LIN {X -0.131,Y -388.858,Z 1048.466,A 0.000,B 0.000,C 90.000,E1 83.856} C_DIS
LIN {X -0.049,Y -379.523,Z 1048.456,A 0.000,B 0.000,C 90.000,E1 82.129} C_DIS
LIN {X -0.037,Y -369.873,Z 1048.447,A 0.000,B 0.000,C 90.000,E1 80.387} C_DIS
LIN {X -0.127,Y -359.894,Z 1048.437,A 0.000,B 0.000,C 90.000,E1 78.634} C_DIS
LIN {X -0.097,Y -346.570,Z 1048.423,A 0.000,B 0.000,C 90.000,E1 76.228} C_DIS
LIN {X 0.098,Y -333.515,Z 1048.410,A 0.000,B 0.000,C 90.000,E1 73.740} C_DIS
LIN {X -0.157,Y -321.006,Z 1048.396,A 0.000,B 0.000,C 90.000,E1 71.275} C_DIS
LIN {X 0.091,Y -308.881,Z 1048.382,A 0.000,B 0.000,C 90.000,E1 68.666} C_DIS
LIN {X 0.079,Y -297.203,Z 1048.367,A 0.000,B 0.000,C 90.000,E1 66.049} C_DIS
LIN {X 0.032,Y -285.773,Z 1048.352,A 0.000,B 0.000,C 90.000,E1 63.384} C_DIS
LIN {X 0.014,Y -275.986,Z 1048.339,A 0.000,B 0.000,C 90.000,E1 61.001} C_DIS
LIN {X 0.100,Y -265.051,Z 1048.323,A 0.000,B 0.000,C 90.000,E1 58.201} C_DIS
LIN {X -0.025,Y -254.368,Z 1048.308,A 0.000,B 0.000,C 90.000,E1 55.388} C_DIS
LIN {X 0.027,Y -242.843,Z 1048.290,A 0.000,B 0.000,C 90.000,E1 52.110} C_DIS
LIN {X 0.019,Y -231.988,Z 1048.271,A 0.000,B 0.000,C 90.000,E1 48.771} C_DIS
LIN {X 0.057,Y -223.046,Z 1048.254,A 0.000,B 0.000,C 90.000,E1 45.729} C_DIS
LIN {X -0.100,Y -214.640,Z 1048.237,A 0.000,B 0.000,C 90.000,E1 42.690} C_DIS
LIN {X 0.029,Y -206.684,Z 1048.220,A 0.000,B 0.000,C 90.000,E1 39.519} C_DIS
LIN {X -0.019,Y -199.257,Z 1048.202,A 0.000,B 0.000,C 90.000,E1 36.343} C_DIS
LIN {X 0.034,Y -192.371,Z 1048.184,A 0.000,B 0.000,C 90.000,E1 33.086} C_DIS
LIN {X 0.034,Y -186.264,Z 1048.166,A 0.000,B 0.000,C 90.000,E1 29.795} C_DIS
LIN {X -0.060,Y -180.873,Z 1048.147,A 0.000,B 0.000,C 90.000,E1 26.488} C_DIS
LIN {X 0.044,Y -176.216,Z 1048.128,A 0.000,B 0.000,C 90.000,E1 23.078} C_DIS
LIN {X -0.014,Y -172.265,Z 1048.109,A 0.000,B 0.000,C 90.000,E1 19.685} C_DIS
LIN {X 0.002,Y -168.389,Z 1048.085,A 0.000,B 0.000,C 90.000,E1 15.371} C_DIS
LIN {X 0.054,Y -165.557,Z 1048.061,A 0.000,B 0.000,C 90.000,E1 11.007} C_DIS
LIN {X 0.024,Y -163.209,Z 1048.022,A 0.000,B 0.000,C 90.000,E1 4.012} C_DIS
LIN {X -0.037,Y -164.388,Z 1047.963,A 0.000,B 0.000,C 90.000,E1 353.394} C_DIS
LIN {X 0.040,Y -167.026,Z 1047.934,A 0.000,B 0.000,C 90.000,E1 348.117} C_DIS
LIN {X -0.032,Y -170.462,Z 1047.910,A 0.000,B 0.000,C 90.000,E1 343.795} C_DIS
LIN {X 0.052,Y -173.950,Z 1047.891,A 0.000,B 0.000,C 90.000,E1 340.315} C_DIS
LIN {X -0.037,Y -178.137,Z 1047.872,A 0.000,B 0.000,C 90.000,E1 336.922} C_DIS
LIN {X 0.030,Y -183.098,Z 1047.853,A 0.000,B 0.000,C 90.000,E1 333.512} C_DIS
LIN {X -0.111,Y -188.880,Z 1047.834,A 0.000,B 0.000,C 90.000,E1 330.205} C_DIS
LIN {X 0.110,Y -195.450,Z 1047.816,A 0.000,B 0.000,C 90.000,E1 326.834} C_DIS
LIN {X -0.044,Y -202.808,Z 1047.798,A 0.000,B 0.000,C 90.000,E1 323.623} C_DIS
LIN {X -0.102,Y -210.701,Z 1047.780,A 0.000,B 0.000,C 90.000,E1 320.436} C_DIS
LIN {X 0.062,Y -220.389,Z 1047.760,A 0.000,B 0.000,C 90.000,E1 316.863} C_DIS
LIN {X 0.075,Y -229.831,Z 1047.743,A 0.000,B 0.000,C 90.000,E1 313.785} C_DIS
LIN {X 0.089,Y -237.669,Z 1047.731,A 0.000,B 0.000,C 90.000,E1 311.515} C_DIS
LIN {X 0.122,Y -246.397,Z 1047.718,A 0.000,B 0.000,C 90.000,E1 309.277} C_DIS
LIN {X 0.137,Y -252.982,Z 1047.710,A 0.000,B 0.000,C 90.000,E1 307.810} C_DIS
LIN {X -0.043,Y -267.797,Z 1047.694,A 0.000,B 0.000,C 90.000,E1 304.978} C_DIS
LIN {X 0.188,Y -286.229,Z 1047.677,A 0.000,B 0.000,C 90.000,E1 301.799} C_DIS
LIN {X -0.040,Y -305.957,Z 1047.660,A 0.000,B 0.000,C 90.000,E1 298.821} C_DIS
LIN {X -0.024,Y -322.578,Z 1047.647,A 0.000,B 0.000,C 90.000,E1 296.539} C_DIS
LIN {X -0.116,Y -332.909,Z 1047.640,A 0.000,B 0.000,C 90.000,E1 295.283} C_DIS
LIN {X -0.126,Y -346.134,Z 1047.632,A 0.000,B 0.000,C 90.000,E1 293.823} C_DIS
LIN {X -0.132,Y -370.998,Z 1047.619,A 0.000,B 0.000,C 90.000,E1 291.408} C_DIS
LIN {X -0.018,Y -390.288,Z 1047.609,A 0.000,B 0.000,C 90.000,E1 289.685} C_DIS
LIN {X 0.047,Y -403.946,Z 1047.603,A 0.000,B 0.000,C 90.000,E1 288.489} C_DIS
LIN {X 0.095,Y -414.628,Z 1047.597,A 0.000,B 0.000,C 90.000,E1 287.528} C_DIS
LIN {X 0.179,Y -422.149,Z 1047.594,A 0.000,B 0.000,C 90.000,E1 286.804} C_DIS
LIN {X -0.051,Y -429.627,Z 1047.589,A 0.000,B 0.000,C 90.000,E1 286.079} C_DIS
LIN {X -0.120,Y -436.988,Z 1047.585,A 0.000,B 0.000,C 90.000,E1 285.300} C_DIS
LIN {X 0.068,Y -444.139,Z 1047.580,A 0.000,B 0.000,C 90.000,E1 284.481} C_DIS
LIN {X -0.013,Y -450.801,Z 1047.576,A 0.000,B 0.000,C 90.000,E1 283.703} C_DIS
LIN {X -0.156,Y -456.953,Z 1047.572,A 0.000,B 0.000,C 90.000,E1 282.939} C_DIS
LIN {X 0.213,Y -462.516,Z 1047.568,A 0.000,B 0.000,C 90.000,E1 282.119} C_DIS
LIN {X 0.084,Y -467.494,Z 1047.563,A 0.000,B 0.000,C 90.000,E1 281.366} C_DIS
LIN {X 0.095,Y -471.818,Z 1047.559,A 0.000,B 0.000,C 90.000,E1 280.602} C_DIS
LIN {X 0.053,Y -475.532,Z 1047.555,A 0.000,B 0.000,C 90.000,E1 279.849} C_DIS
LIN {X 0.255,Y -477.654,Z 1047.552,A 0.000,B 0.000,C 90.000,E1 279.321} C_DIS
LIN {X -0.079,Y -479.547,Z 1047.549,A 0.000,B 0.000,C 90.000,E1 278.859} C_DIS
LIN {X -0.183,Y -482.701,Z 1047.544,A 0.000,B 0.000,C 90.000,E1 277.871} C_DIS
LIN {X -0.016,Y -484.005,Z 1047.541,A 0.000,B 0.000,C 90.000,E1 277.352} C_DIS
LIN {X 0.164,Y -485.073,Z 1047.538,A 0.000,B 0.000,C 90.000,E1 276.834} C_DIS
LIN {X -0.132,Y -485.850,Z 1047.535,A 0.000,B 0.000,C 90.000,E1 276.372} C_DIS
LIN {X 0.060,Y -486.341,Z 1047.533,A 0.000,B 0.000,C 90.000,E1 275.853} C_DIS
LIN {X 0.257,Y -486.480,Z 1047.530,A 0.000,B 0.000,C 90.000,E1 275.334} C_DIS
LIN {X -0.071,Y -486.178,Z 1047.527,A 0.000,B 0.000,C 90.000,E1 274.878} C_DIS
LIN {X 0.129,Y -485.411,Z 1047.524,A 0.000,B 0.000,C 90.000,E1 274.359} C_DIS
LIN {X -0.159,Y -484.101,Z 1047.522,A 0.000,B 0.000,C 90.000,E1 273.898} C_DIS
LIN {X 0.001,Y -482.154,Z 1047.519,A 0.000,B 0.000,C 90.000,E1 273.383} C_DIS
LIN {X 0.179,Y -479.498,Z 1047.516,A 0.000,B 0.000,C 90.000,E1 272.865} C_DIS
LIN {X -0.163,Y -476.100,Z 1047.513,A 0.000,B 0.000,C 90.000,E1 272.407} C_DIS
LIN {X -0.041,Y -471.794,Z 1047.510,A 0.000,B 0.000,C 90.000,E1 271.892} C_DIS
LIN {X 0.070,Y -466.518,Z 1047.508,A 0.000,B 0.000,C 90.000,E1 271.375} C_DIS
LIN {X -0.007,Y -460.835,Z 1047.505,A 0.000,B 0.000,C 90.000,E1 270.917} C_DIS
LIN {X 0.220,Y -454.718,Z 1047.503,A 0.000,B 0.000,C 90.000,E1 270.458} C_DIS
LIN {X -0.065,Y -448.087,Z 1047.501,A 0.000,B 0.000,C 90.000,E1 270.115} C_DIS
LIN {X 0.112,Y -440.719,Z 1047.499,A 0.000,B 0.000,C 90.000,E1 269.771} C_DIS
LIN {X -0.035,Y -432.780,Z 1047.497,A 0.000,B 0.000,C 90.000,E1 269.542} C_DIS
LIN {X -0.102,Y -424.050,Z 1047.496,A 0.000,B 0.000,C 90.000,E1 269.370} C_DIS
LIN {X -0.035,Y -411.377,Z 1047.495,A 0.000,B 0.000,C 90.000,E1 269.198} C_DIS
LIN {X -0.063,Y -401.436,Z 1047.495,A 0.000,B 0.000,C 90.000,E1 269.141} C_DIS
LIN {X 0.162,Y -392.391,Z 1047.495,A 0.000,B 0.000,C 90.000,E1 269.083} C_DIS
LIN {X 0.049,Y -181.341,Z 1047.495,A 0.000,B 0.000,C 90.000,E1 269.083} C_DIS
LIN {X 0.081,Y -180.907,Z 1047.474,A 0.000,B 0.000,C 90.000,E1 265.355} C_DIS
LIN {X -0.026,Y -180.694,Z 1047.470,A 0.000,B 0.000,C 90.000,E1 264.546} C_DIS
LIN {X 0.052,Y -178.779,Z 1047.442,A 0.000,B 0.000,C 90.000,E1 259.454} C_DIS
LIN {X -0.045,Y -175.825,Z 1047.413,A 0.000,B 0.000,C 90.000,E1 254.393} C_DIS
LIN {X -0.044,Y -172.014,Z 1047.385,A 0.000,B 0.000,C 90.000,E1 249.263} C_DIS
LIN {X -0.068,Y -171.434,Z 1047.380,A 0.000,B 0.000,C 90.000,E1 248.411} C_DIS
LIN {X -0.013,Y -167.670,Z 1047.356,A 0.000,B 0.000,C 90.000,E1 244.076} C_DIS
LIN {X -0.073,Y -166.344,Z 1047.346,A 0.000,B 0.000,C 90.000,E1 242.359} C_DIS
LIN {X -0.080,Y -163.079,Z 1047.327,A 0.000,B 0.000,C 90.000,E1 238.869} C_DIS
LIN {X -0.029,Y -161.020,Z 1047.312,A 0.000,B 0.000,C 90.000,E1 236.215} C_DIS
LIN {X -0.045,Y -157.762,Z 1047.293,A 0.000,B 0.000,C 90.000,E1 232.683} C_DIS
LIN {X 0.019,Y -155.800,Z 1047.278,A 0.000,B 0.000,C 90.000,E1 229.989} C_DIS
LIN {X 0.073,Y -152.052,Z 1047.253,A 0.000,B 0.000,C 90.000,E1 225.486} C_DIS
LIN {X -0.020,Y -150.303,Z 1047.238,A 0.000,B 0.000,C 90.000,E1 222.813} C_DIS
LIN {X 0.016,Y -147.048,Z 1047.213,A 0.000,B 0.000,C 90.000,E1 218.257} C_DIS
LIN {X 0.008,Y -145.627,Z 1047.197,A 0.000,B 0.000,C 90.000,E1 215.518} C_DIS
LIN {X 0.007,Y -143.010,Z 1047.172,A 0.000,B 0.000,C 90.000,E1 210.924} C_DIS
LIN {X -0.062,Y -141.637,Z 1047.151,A 0.000,B 0.000,C 90.000,E1 207.257} C_DIS
LIN {X -0.011,Y -139.438,Z 1047.115,A 0.000,B 0.000,C 90.000,E1 200.737} C_DIS
LIN {X 0.042,Y -139.170,Z 1047.105,A 0.000,B 0.000,C 90.000,E1 198.852} C_DIS
LIN {X -0.060,Y -138.318,Z 1047.053,A 0.000,B 0.000,C 90.000,E1 189.557} C_DIS
LIN {X -0.052,Y -139.474,Z 1047.006,A 0.000,B 0.000,C 90.000,E1 181.146} C_DIS
LIN {X 0.029,Y -141.050,Z 1046.975,A 0.000,B 0.000,C 90.000,E1 175.527} C_DIS
LIN {X -0.018,Y -142.421,Z 1046.960,A 0.000,B 0.000,C 90.000,E1 172.761} C_DIS
LIN {X 0.044,Y -144.657,Z 1046.934,A 0.000,B 0.000,C 90.000,E1 168.117} C_DIS
LIN {X -0.038,Y -147.853,Z 1046.909,A 0.000,B 0.000,C 90.000,E1 163.559} C_DIS
LIN {X 0.046,Y -150.555,Z 1046.888,A 0.000,B 0.000,C 90.000,E1 159.880} C_DIS
LIN {X -0.015,Y -154.022,Z 1046.868,A 0.000,B 0.000,C 90.000,E1 156.282} C_DIS
LIN {X -0.017,Y -157.438,Z 1046.848,A 0.000,B 0.000,C 90.000,E1 152.692} C_DIS
LIN {X 0.004,Y -161.652,Z 1046.828,A 0.000,B 0.000,C 90.000,E1 149.125} C_DIS
LIN {X 0.021,Y -165.848,Z 1046.809,A 0.000,B 0.000,C 90.000,E1 145.595} C_DIS
LIN {X 0.013,Y -170.823,Z 1046.790,A 0.000,B 0.000,C 90.000,E1 142.110} C_DIS
LIN {X -0.071,Y -175.692,Z 1046.770,A 0.000,B 0.000,C 90.000,E1 138.690} C_DIS
LIN {X 0.053,Y -181.305,Z 1046.751,A 0.000,B 0.000,C 90.000,E1 135.243} C_DIS
LIN {X -0.075,Y -186.786,Z 1046.733,A 0.000,B 0.000,C 90.000,E1 131.919} C_DIS
LIN {X -0.005,Y -191.379,Z 1046.719,A 0.000,B 0.000,C 90.000,E1 129.402} C_DIS
LIN {X -0.055,Y -197.607,Z 1046.700,A 0.000,B 0.000,C 90.000,E1 125.931} C_DIS
LIN {X 0.103,Y -197.923,Z 1046.699,A 0.000,B 0.000,C 90.000,E1 125.724} C_DIS
LIN {X 0.116,Y -304.006,Z 1046.699,A 0.000,B 0.000,C 90.000,E1 125.724} C_DIS
LIN {X 0.033,Y -305.067,Z 1046.698,A 0.000,B 0.000,C 90.000,E1 125.724} C_DIS
LIN {X -0.019,Y -310.030,Z 1046.697,A 0.000,B 0.000,C 90.000,E1 125.518} C_DIS
LIN {X -0.072,Y -312.622,Z 1046.696,A 0.000,B 0.000,C 90.000,E1 125.311} C_DIS
LIN {X -0.036,Y -316.422,Z 1046.693,A 0.000,B 0.000,C 90.000,E1 124.818} C_DIS
LIN {X 0.019,Y -318.184,Z 1046.692,A 0.000,B 0.000,C 90.000,E1 124.485} C_DIS
LIN {X -0.188,Y -319.561,Z 1046.690,A 0.000,B 0.000,C 90.000,E1 124.199} C_DIS
LIN {X 0.022,Y -332.011,Z 1046.670,A 0.000,B 0.000,C 90.000,E1 120.669} C_DIS
LIN {X -0.149,Y -343.638,Z 1046.655,A 0.000,B 0.000,C 90.000,E1 117.897} C_DIS
LIN {X -0.168,Y -356.702,Z 1046.640,A 0.000,B 0.000,C 90.000,E1 115.155} C_DIS
LIN {X -0.193,Y -369.617,Z 1046.626,A 0.000,B 0.000,C 90.000,E1 112.770} C_DIS
LIN {X -0.183,Y -383.852,Z 1046.613,A 0.000,B 0.000,C 90.000,E1 110.429} C_DIS
LIN {X -0.076,Y -399.507,Z 1046.601,A 0.000,B 0.000,C 90.000,E1 108.127} C_DIS
LIN {X -0.086,Y -416.693,Z 1046.588,A 0.000,B 0.000,C 90.000,E1 105.898} C_DIS
LIN {X -0.011,Y -435.533,Z 1046.576,A 0.000,B 0.000,C 90.000,E1 103.716} C_DIS
LIN {X 0.048,Y -455.539,Z 1046.565,A 0.000,B 0.000,C 90.000,E1 101.658} C_DIS
LIN {X -0.173,Y -468.201,Z 1046.558,A 0.000,B 0.000,C 90.000,E1 100.489} C_DIS
LIN {X -0.225,Y -470.121,Z 1046.557,A 0.000,B 0.000,C 90.000,E1 100.254} C_DIS
LIN {X 0.188,Y -471.578,Z 1046.555,A 0.000,B 0.000,C 90.000,E1 99.962} C_DIS
LIN {X -0.181,Y -473.559,Z 1046.553,A 0.000,B 0.000,C 90.000,E1 99.500} C_DIS
LIN {X 0.002,Y -474.416,Z 1046.550,A 0.000,B 0.000,C 90.000,E1 98.973} C_DIS
LIN {X 0.121,Y -474.297,Z 1046.547,A 0.000,B 0.000,C 90.000,E1 98.454} C_DIS
LIN {X -0.220,Y -473.191,Z 1046.544,A 0.000,B 0.000,C 90.000,E1 97.992} C_DIS
LIN {X 0.110,Y -472.216,Z 1046.543,A 0.000,B 0.000,C 90.000,E1 97.701} C_DIS
LIN {X -0.030,Y -470.902,Z 1046.542,A 0.000,B 0.000,C 90.000,E1 97.466} C_DIS
LIN {X 0.025,Y -458.510,Z 1046.532,A 0.000,B 0.000,C 90.000,E1 95.682} C_DIS
LIN {X 0.035,Y -444.230,Z 1046.520,A 0.000,B 0.000,C 90.000,E1 93.612} C_DIS
LIN {X 0.127,Y -430.922,Z 1046.508,A 0.000,B 0.000,C 90.000,E1 91.489} C_DIS
LIN {X 0.104,Y -415.490,Z 1046.493,A 0.000,B 0.000,C 90.000,E1 88.797} C_DIS
LIN {X -0.121,Y -405.344,Z 1046.483,A 0.000,B 0.000,C 90.000,E1 86.906} C_DIS
LIN {X -0.103,Y -394.835,Z 1046.472,A 0.000,B 0.000,C 90.000,E1 84.951} C_DIS
LIN {X 0.092,Y -385.623,Z 1046.462,A 0.000,B 0.000,C 90.000,E1 83.223} C_DIS
LIN {X 0.158,Y -376.191,Z 1046.453,A 0.000,B 0.000,C 90.000,E1 81.489} C_DIS
LIN {X 0.109,Y -366.399,Z 1046.443,A 0.000,B 0.000,C 90.000,E1 79.746} C_DIS
LIN {X -0.046,Y -356.389,Z 1046.433,A 0.000,B 0.000,C 90.000,E1 77.993} C_DIS
LIN {X -0.025,Y -343.128,Z 1046.420,A 0.000,B 0.000,C 90.000,E1 75.574} C_DIS
LIN {X -0.077,Y -327.078,Z 1046.403,A 0.000,B 0.000,C 90.000,E1 72.489} C_DIS
LIN {X 0.024,Y -314.747,Z 1046.389,A 0.000,B 0.000,C 90.000,E1 69.934} C_DIS
LIN {X -0.164,Y -301.401,Z 1046.372,A 0.000,B 0.000,C 90.000,E1 67.050} C_DIS
LIN {X 0.037,Y -289.864,Z 1046.358,A 0.000,B 0.000,C 90.000,E1 64.357} C_DIS
LIN {X 0.101,Y -280.007,Z 1046.344,A 0.000,B 0.000,C 90.000,E1 61.975} C_DIS
LIN {X 0.148,Y -268.942,Z 1046.329,A 0.000,B 0.000,C 90.000,E1 59.203} C_DIS
LIN {X 0.078,Y -259.487,Z 1046.315,A 0.000,B 0.000,C 90.000,E1 56.755} C_DIS
LIN {X -0.034,Y -248.987,Z 1046.299,A 0.000,B 0.000,C 90.000,E1 53.909} C_DIS
LIN {X 0.011,Y -237.704,Z 1046.281,A 0.000,B 0.000,C 90.000,E1 50.598} C_DIS
LIN {X -0.015,Y -227.230,Z 1046.262,A 0.000,B 0.000,C 90.000,E1 47.229} C_DIS
LIN {X -0.083,Y -218.586,Z 1046.245,A 0.000,B 0.000,C 90.000,E1 44.190} C_DIS
LIN {X -0.035,Y -210.398,Z 1046.228,A 0.000,B 0.000,C 90.000,E1 41.067} C_DIS
LIN {X 0.013,Y -202.682,Z 1046.211,A 0.000,B 0.000,C 90.000,E1 37.890} C_DIS
LIN {X -0.053,Y -195.526,Z 1046.193,A 0.000,B 0.000,C 90.000,E1 34.692} C_DIS
LIN {X 0.059,Y -190.552,Z 1046.179,A 0.000,B 0.000,C 90.000,E1 32.212} C_DIS
LIN {X -0.076,Y -184.618,Z 1046.161,A 0.000,B 0.000,C 90.000,E1 28.949} C_DIS
LIN {X -0.045,Y -179.416,Z 1046.142,A 0.000,B 0.000,C 90.000,E1 25.591} C_DIS
LIN {X -0.051,Y -174.963,Z 1046.123,A 0.000,B 0.000,C 90.000,E1 22.206} C_DIS
LIN {X -0.037,Y -171.220,Z 1046.104,A 0.000,B 0.000,C 90.000,E1 18.779} C_DIS
LIN {X -0.097,Y -167.530,Z 1046.080,A 0.000,B 0.000,C 90.000,E1 14.481} C_DIS
LIN {X 0.055,Y -165.004,Z 1046.056,A 0.000,B 0.000,C 90.000,E1 10.074} C_DIS
LIN {X -0.038,Y -162.952,Z 1046.017,A 0.000,B 0.000,C 90.000,E1 3.094} C_DIS
LIN {X -0.042,Y -164.283,Z 1045.963,A 0.000,B 0.000,C 90.000,E1 353.394} C_DIS
LIN {X 0.031,Y -166.926,Z 1045.934,A 0.000,B 0.000,C 90.000,E1 348.117} C_DIS
LIN {X -0.044,Y -170.370,Z 1045.910,A 0.000,B 0.000,C 90.000,E1 343.795} C_DIS
LIN {X 0.037,Y -173.856,Z 1045.891,A 0.000,B 0.000,C 90.000,E1 340.315} C_DIS
LIN {X -0.054,Y -178.038,Z 1045.872,A 0.000,B 0.000,C 90.000,E1 336.922} C_DIS
LIN {X 0.010,Y -183.000,Z 1045.853,A 0.000,B 0.000,C 90.000,E1 333.512} C_DIS
LIN {X 0.125,Y -188.808,Z 1045.834,A 0.000,B 0.000,C 90.000,E1 330.127} C_DIS
LIN {X 0.084,Y -195.389,Z 1045.816,A 0.000,B 0.000,C 90.000,E1 326.834} C_DIS
LIN {X -0.072,Y -202.763,Z 1045.798,A 0.000,B 0.000,C 90.000,E1 323.623} C_DIS
LIN {X -0.132,Y -210.641,Z 1045.780,A 0.000,B 0.000,C 90.000,E1 320.436} C_DIS
LIN {X 0.028,Y -220.328,Z 1045.760,A 0.000,B 0.000,C 90.000,E1 316.863} C_DIS
LIN {X 0.038,Y -229.752,Z 1045.743,A 0.000,B 0.000,C 90.000,E1 313.785} C_DIS
LIN {X 0.049,Y -237.577,Z 1045.731,A 0.000,B 0.000,C 90.000,E1 311.515} C_DIS
LIN {X 0.080,Y -246.318,Z 1045.718,A 0.000,B 0.000,C 90.000,E1 309.277} C_DIS
LIN {X 0.092,Y -252.891,Z 1045.710,A 0.000,B 0.000,C 90.000,E1 307.810} C_DIS
LIN {X 0.061,Y -267.723,Z 1045.694,A 0.000,B 0.000,C 90.000,E1 304.945} C_DIS
LIN {X 0.132,Y -286.216,Z 1045.677,A 0.000,B 0.000,C 90.000,E1 301.799} C_DIS
LIN {X -0.099,Y -305.987,Z 1045.660,A 0.000,B 0.000,C 90.000,E1 298.821} C_DIS
LIN {X -0.085,Y -322.667,Z 1045.647,A 0.000,B 0.000,C 90.000,E1 296.539} C_DIS
LIN {X 0.073,Y -335.551,Z 1045.639,A 0.000,B 0.000,C 90.000,E1 294.951} C_DIS
LIN {X -0.083,Y -349.150,Z 1045.631,A 0.000,B 0.000,C 90.000,E1 293.515} C_DIS
LIN {X 0.198,Y -379.470,Z 1045.615,A 0.000,B 0.000,C 90.000,E1 290.610} C_DIS
LIN {X -0.047,Y -395.869,Z 1045.607,A 0.000,B 0.000,C 90.000,E1 289.214} C_DIS
LIN {X 0.126,Y -406.758,Z 1045.601,A 0.000,B 0.000,C 90.000,E1 288.236} C_DIS
LIN {X 0.173,Y -414.756,Z 1045.597,A 0.000,B 0.000,C 90.000,E1 287.511} C_DIS
LIN {X -0.038,Y -422.492,Z 1045.593,A 0.000,B 0.000,C 90.000,E1 286.804} C_DIS
LIN {X 0.076,Y -429.992,Z 1045.589,A 0.000,B 0.000,C 90.000,E1 286.024} C_DIS
LIN {X 0.172,Y -439.780,Z 1045.583,A 0.000,B 0.000,C 90.000,E1 284.954} C_DIS
LIN {X 0.056,Y -446.756,Z 1045.579,A 0.000,B 0.000,C 90.000,E1 284.175} C_DIS
LIN {X -0.120,Y -453.230,Z 1045.574,A 0.000,B 0.000,C 90.000,E1 283.411} C_DIS
LIN {X 0.213,Y -459.118,Z 1045.570,A 0.000,B 0.000,C 90.000,E1 282.591} C_DIS
LIN {X 0.149,Y -464.473,Z 1045.566,A 0.000,B 0.000,C 90.000,E1 281.827} C_DIS
LIN {X 0.042,Y -469.238,Z 1045.562,A 0.000,B 0.000,C 90.000,E1 281.074} C_DIS
LIN {X 0.064,Y -473.345,Z 1045.557,A 0.000,B 0.000,C 90.000,E1 280.310} C_DIS
LIN {X 0.039,Y -476.856,Z 1045.553,A 0.000,B 0.000,C 90.000,E1 279.557} C_DIS
LIN {X 0.043,Y -479.763,Z 1045.549,A 0.000,B 0.000,C 90.000,E1 278.803} C_DIS
LIN {X -0.056,Y -482.894,Z 1045.543,A 0.000,B 0.000,C 90.000,E1 277.814} C_DIS
LIN {X 0.113,Y -484.162,Z 1045.541,A 0.000,B 0.000,C 90.000,E1 277.296} C_DIS
LIN {X -0.187,Y -485.227,Z 1045.538,A 0.000,B 0.000,C 90.000,E1 276.834} C_DIS
LIN {X 0.001,Y -486.001,Z 1045.535,A 0.000,B 0.000,C 90.000,E1 276.315} C_DIS
LIN {X 0.194,Y -486.460,Z 1045.532,A 0.000,B 0.000,C 90.000,E1 275.796} C_DIS
LIN {X -0.092,Y -486.565,Z 1045.530,A 0.000,B 0.000,C 90.000,E1 275.334} C_DIS
LIN {X 0.065,Y -486.236,Z 1045.527,A 0.000,B 0.000,C 90.000,E1 274.821} C_DIS
LIN {X -0.217,Y -485.456,Z 1045.524,A 0.000,B 0.000,C 90.000,E1 274.359} C_DIS
LIN {X -0.022,Y -484.097,Z 1045.521,A 0.000,B 0.000,C 90.000,E1 273.841} C_DIS
LIN {X 0.138,Y -482.101,Z 1045.519,A 0.000,B 0.000,C 90.000,E1 273.326} C_DIS
LIN {X -0.163,Y -479.410,Z 1045.516,A 0.000,B 0.000,C 90.000,E1 272.865} C_DIS
LIN {X 0.143,Y -477.802,Z 1045.514,A 0.000,B 0.000,C 90.000,E1 272.579} C_DIS
LIN {X -0.203,Y -473.886,Z 1045.512,A 0.000,B 0.000,C 90.000,E1 272.121} C_DIS
LIN {X -0.080,Y -469.073,Z 1045.509,A 0.000,B 0.000,C 90.000,E1 271.604} C_DIS
LIN {X 0.187,Y -463.534,Z 1045.506,A 0.000,B 0.000,C 90.000,E1 271.088} C_DIS
LIN {X -0.157,Y -457.703,Z 1045.504,A 0.000,B 0.000,C 90.000,E1 270.688} C_DIS
LIN {X -0.161,Y -451.404,Z 1045.501,A 0.000,B 0.000,C 90.000,E1 270.286} C_DIS
LIN {X 0.157,Y -447.914,Z 1045.500,A 0.000,B 0.000,C 90.000,E1 270.057} C_DIS
LIN {X -0.092,Y -440.528,Z 1045.499,A 0.000,B 0.000,C 90.000,E1 269.771} C_DIS
LIN {X -0.157,Y -436.976,Z 1045.498,A 0.000,B 0.000,C 90.000,E1 269.656} C_DIS
LIN {X -0.006,Y -428.802,Z 1045.497,A 0.000,B 0.000,C 90.000,E1 269.427} C_DIS
LIN {X 0.200,Y -420.015,Z 1045.496,A 0.000,B 0.000,C 90.000,E1 269.255} C_DIS
LIN {X -0.133,Y -411.331,Z 1045.495,A 0.000,B 0.000,C 90.000,E1 269.198} C_DIS
LIN {X -0.158,Y -401.181,Z 1045.495,A 0.000,B 0.000,C 90.000,E1 269.141} C_DIS
LIN {X 0.129,Y -395.536,Z 1045.495,A 0.000,B 0.000,C 90.000,E1 269.083} C_DIS
LIN {X 0.033,Y -181.340,Z 1045.495,A 0.000,B 0.000,C 90.000,E1 269.083} C_DIS
LIN {X 0.040,Y -180.906,Z 1045.474,A 0.000,B 0.000,C 90.000,E1 265.355} C_DIS
LIN {X -0.066,Y -180.688,Z 1045.470,A 0.000,B 0.000,C 90.000,E1 264.546} C_DIS
LIN {X 0.012,Y -178.772,Z 1045.441,A 0.000,B 0.000,C 90.000,E1 259.454} C_DIS
LIN {X 0.084,Y -175.818,Z 1045.413,A 0.000,B 0.000,C 90.000,E1 254.338} C_DIS
LIN {X 0.078,Y -172.006,Z 1045.385,A 0.000,B 0.000,C 90.000,E1 249.209} C_DIS
LIN {X 0.052,Y -171.423,Z 1045.380,A 0.000,B 0.000,C 90.000,E1 248.358} C_DIS
LIN {X -0.052,Y -167.661,Z 1045.356,A 0.000,B 0.000,C 90.000,E1 244.076} C_DIS
LIN {X 0.036,Y -166.330,Z 1045.346,A 0.000,B 0.000,C 90.000,E1 242.308} C_DIS
LIN {X 0.022,Y -163.068,Z 1045.327,A 0.000,B 0.000,C 90.000,E1 238.820} C_DIS
LIN {X -0.067,Y -161.007,Z 1045.312,A 0.000,B 0.000,C 90.000,E1 236.215} C_DIS
LIN {X 0.044,Y -157.751,Z 1045.292,A 0.000,B 0.000,C 90.000,E1 232.637} C_DIS
LIN {X -0.018,Y -155.789,Z 1045.278,A 0.000,B 0.000,C 90.000,E1 229.989} C_DIS
LIN {X 0.037,Y -152.043,Z 1045.253,A 0.000,B 0.000,C 90.000,E1 225.486} C_DIS
LIN {X 0.054,Y -150.292,Z 1045.238,A 0.000,B 0.000,C 90.000,E1 222.771} C_DIS
LIN {X -0.020,Y -147.040,Z 1045.213,A 0.000,B 0.000,C 90.000,E1 218.257} C_DIS
LIN {X -0.027,Y -145.620,Z 1045.197,A 0.000,B 0.000,C 90.000,E1 215.518} C_DIS
LIN {X -0.029,Y -143.004,Z 1045.172,A 0.000,B 0.000,C 90.000,E1 210.924} C_DIS
LIN {X 0.029,Y -141.630,Z 1045.151,A 0.000,B 0.000,C 90.000,E1 207.206} C_DIS
LIN {X -0.045,Y -139.435,Z 1045.115,A 0.000,B 0.000,C 90.000,E1 200.737} C_DIS
LIN {X 0.009,Y -139.167,Z 1045.105,A 0.000,B 0.000,C 90.000,E1 198.852} C_DIS
LIN {X 0.042,Y -138.316,Z 1045.053,A 0.000,B 0.000,C 90.000,E1 189.500} C_DIS
LIN {X 0.053,Y -139.475,Z 1045.006,A 0.000,B 0.000,C 90.000,E1 181.088} C_DIS
LIN {X -0.006,Y -141.056,Z 1044.975,A 0.000,B 0.000,C 90.000,E1 175.527} C_DIS
LIN {X -0.052,Y -142.429,Z 1044.960,A 0.000,B 0.000,C 90.000,E1 172.761} C_DIS
LIN {X 0.009,Y -144.665,Z 1044.934,A 0.000,B 0.000,C 90.000,E1 168.117} C_DIS
LIN {X -0.007,Y -147.250,Z 1044.914,A 0.000,B 0.000,C 90.000,E1 164.448} C_DIS
LIN {X 0.010,Y -150.567,Z 1044.888,A 0.000,B 0.000,C 90.000,E1 159.880} C_DIS
LIN {X 0.090,Y -154.036,Z 1044.868,A 0.000,B 0.000,C 90.000,E1 156.230} C_DIS
LIN {X 0.018,Y -157.452,Z 1044.848,A 0.000,B 0.000,C 90.000,E1 152.666} C_DIS
LIN {X -0.034,Y -161.670,Z 1044.828,A 0.000,B 0.000,C 90.000,E1 149.125} C_DIS
LIN {X -0.017,Y -165.866,Z 1044.809,A 0.000,B 0.000,C 90.000,E1 145.595} C_DIS
LIN {X -0.025,Y -170.843,Z 1044.789,A 0.000,B 0.000,C 90.000,E1 142.110} C_DIS
LIN {X 0.021,Y -175.712,Z 1044.770,A 0.000,B 0.000,C 90.000,E1 138.647} C_DIS
LIN {X 0.013,Y -181.324,Z 1044.751,A 0.000,B 0.000,C 90.000,E1 135.243} C_DIS
LIN {X 0.007,Y -186.809,Z 1044.733,A 0.000,B 0.000,C 90.000,E1 131.881} C_DIS
LIN {X -0.047,Y -191.398,Z 1044.719,A 0.000,B 0.000,C 90.000,E1 129.402} C_DIS
LIN {X 0.063,Y -197.631,Z 1044.699,A 0.000,B 0.000,C 90.000,E1 125.884} C_DIS
LIN {X -0.034,Y -197.843,Z 1044.699,A 0.000,B 0.000,C 90.000,E1 125.804} C_DIS
LIN {X -0.099,Y -304.134,Z 1044.699,A 0.000,B 0.000,C 90.000,E1 125.804} C_DIS
LIN {X 0.073,Y -310.224,Z 1044.697,A 0.000,B 0.000,C 90.000,E1 125.518} C_DIS
LIN {X -0.140,Y -312.986,Z 1044.696,A 0.000,B 0.000,C 90.000,E1 125.311} C_DIS
LIN {X 0.014,Y -316.737,Z 1044.693,A 0.000,B 0.000,C 90.000,E1 124.771} C_DIS
LIN {X -0.011,Y -318.393,Z 1044.691,A 0.000,B 0.000,C 90.000,E1 124.452} C_DIS
LIN {X 0.120,Y -320.761,Z 1044.688,A 0.000,B 0.000,C 90.000,E1 123.785} C_DIS
LIN {X 0.147,Y -330.924,Z 1044.672,A 0.000,B 0.000,C 90.000,E1 120.924} C_DIS
LIN {X -0.051,Y -342.412,Z 1044.656,A 0.000,B 0.000,C 90.000,E1 118.153} C_DIS
LIN {X -0.106,Y -355.333,Z 1044.641,A 0.000,B 0.000,C 90.000,E1 115.412} C_DIS
LIN {X -0.019,Y -368.109,Z 1044.628,A 0.000,B 0.000,C 90.000,E1 113.003} C_DIS
LIN {X -0.049,Y -382.194,Z 1044.615,A 0.000,B 0.000,C 90.000,E1 110.663} C_DIS
LIN {X 0.014,Y -397.688,Z 1044.602,A 0.000,B 0.000,C 90.000,E1 108.362} C_DIS
LIN {X -0.041,Y -414.699,Z 1044.590,A 0.000,B 0.000,C 90.000,E1 106.134} C_DIS
LIN {X 0.087,Y -433.353,Z 1044.578,A 0.000,B 0.000,C 90.000,E1 103.939} C_DIS
LIN {X -0.020,Y -453.293,Z 1044.566,A 0.000,B 0.000,C 90.000,E1 101.883} C_DIS
LIN {X 0.060,Y -468.424,Z 1044.558,A 0.000,B 0.000,C 90.000,E1 100.433} C_DIS
LIN {X -0.017,Y -470.305,Z 1044.557,A 0.000,B 0.000,C 90.000,E1 100.197} C_DIS
LIN {X -0.094,Y -471.729,Z 1044.555,A 0.000,B 0.000,C 90.000,E1 99.962} C_DIS
LIN {X 0.004,Y -473.627,Z 1044.552,A 0.000,B 0.000,C 90.000,E1 99.443} C_DIS
LIN {X 0.188,Y -474.418,Z 1044.550,A 0.000,B 0.000,C 90.000,E1 98.916} C_DIS
LIN {X -0.160,Y -474.236,Z 1044.547,A 0.000,B 0.000,C 90.000,E1 98.454} C_DIS
LIN {X -0.033,Y -473.061,Z 1044.544,A 0.000,B 0.000,C 90.000,E1 97.936} C_DIS
LIN {X -0.170,Y -472.045,Z 1044.543,A 0.000,B 0.000,C 90.000,E1 97.701} C_DIS
LIN {X 0.157,Y -470.681,Z 1044.541,A 0.000,B 0.000,C 90.000,E1 97.409} C_DIS
LIN {X 0.204,Y -458.264,Z 1044.531,A 0.000,B 0.000,C 90.000,E1 95.625} C_DIS
LIN {X 0.015,Y -445.759,Z 1044.521,A 0.000,B 0.000,C 90.000,E1 93.841} C_DIS
LIN {X -0.036,Y -433.918,Z 1044.511,A 0.000,B 0.000,C 90.000,E1 92.007} C_DIS
LIN {X 0.153,Y -416.757,Z 1044.495,A 0.000,B 0.000,C 90.000,E1 89.026} C_DIS
LIN {X -0.050,Y -406.599,Z 1044.484,A 0.000,B 0.000,C 90.000,E1 87.135} C_DIS
LIN {X -0.072,Y -397.653,Z 1044.475,A 0.000,B 0.000,C 90.000,E1 85.469} C_DIS
LIN {X 0.173,Y -388.511,Z 1044.465,A 0.000,B 0.000,C 90.000,E1 83.742} C_DIS
LIN {X -0.085,Y -379.177,Z 1044.456,A 0.000,B 0.000,C 90.000,E1 82.064} C_DIS
LIN {X -0.131,Y -369.477,Z 1044.446,A 0.000,B 0.000,C 90.000,E1 80.330} C_DIS
LIN {X 0.126,Y -359.515,Z 1044.436,A 0.000,B 0.000,C 90.000,E1 78.522} C_DIS
LIN {X -0.134,Y -347.896,Z 1044.425,A 0.000,B 0.000,C 90.000,E1 76.464} C_DIS
LIN {X 0.095,Y -334.795,Z 1044.411,A 0.000,B 0.000,C 90.000,E1 73.976} C_DIS
LIN {X -0.126,Y -322.231,Z 1044.397,A 0.000,B 0.000,C 90.000,E1 71.511} C_DIS
LIN {X 0.072,Y -308.555,Z 1044.381,A 0.000,B 0.000,C 90.000,E1 68.592} C_DIS
LIN {X 0.059,Y -298.314,Z 1044.368,A 0.000,B 0.000,C 90.000,E1 66.305} C_DIS
LIN {X 0.036,Y -286.843,Z 1044.354,A 0.000,B 0.000,C 90.000,E1 63.640} C_DIS
LIN {X 0.039,Y -277.003,Z 1044.340,A 0.000,B 0.000,C 90.000,E1 61.257} C_DIS
LIN {X 0.012,Y -266.020,Z 1044.325,A 0.000,B 0.000,C 90.000,E1 58.486} C_DIS
LIN {X -0.089,Y -255.303,Z 1044.309,A 0.000,B 0.000,C 90.000,E1 55.674} C_DIS
LIN {X -0.008,Y -243.666,Z 1044.291,A 0.000,B 0.000,C 90.000,E1 52.396} C_DIS
LIN {X 0.008,Y -232.742,Z 1044.273,A 0.000,B 0.000,C 90.000,E1 49.057} C_DIS
LIN {X 0.005,Y -222.645,Z 1044.254,A 0.000,B 0.000,C 90.000,E1 45.648} C_DIS
LIN {X -0.002,Y -214.193,Z 1044.236,A 0.000,B 0.000,C 90.000,E1 42.567} C_DIS
LIN {X -0.040,Y -206.257,Z 1044.219,A 0.000,B 0.000,C 90.000,E1 39.439} C_DIS
LIN {X 0.061,Y -198.801,Z 1044.201,A 0.000,B 0.000,C 90.000,E1 36.217} C_DIS
LIN {X 0.104,Y -191.906,Z 1044.183,A 0.000,B 0.000,C 90.000,E1 32.959} C_DIS
LIN {X 0.093,Y -185.801,Z 1044.165,A 0.000,B 0.000,C 90.000,E1 29.667} C_DIS
LIN {X -0.013,Y -180.423,Z 1044.146,A 0.000,B 0.000,C 90.000,E1 26.360} C_DIS
LIN {X 0.077,Y -175.788,Z 1044.128,A 0.000,B 0.000,C 90.000,E1 22.950} C_DIS
LIN {X -0.051,Y -171.878,Z 1044.109,A 0.000,B 0.000,C 90.000,E1 19.577} C_DIS
LIN {X 0.006,Y -168.013,Z 1044.085,A 0.000,B 0.000,C 90.000,E1 15.245} C_DIS
LIN {X 0.009,Y -165.253,Z 1044.061,A 0.000,B 0.000,C 90.000,E1 10.894} C_DIS
LIN {X 0.019,Y -163.106,Z 1044.026,A 0.000,B 0.000,C 90.000,E1 4.759} C_DIS
LIN {X -0.046,Y -164.184,Z 1043.963,A 0.000,B 0.000,C 90.000,E1 353.394} C_DIS
LIN {X 0.023,Y -166.839,Z 1043.934,A 0.000,B 0.000,C 90.000,E1 348.117} C_DIS
LIN {X -0.054,Y -170.285,Z 1043.910,A 0.000,B 0.000,C 90.000,E1 343.795} C_DIS
LIN {X 0.025,Y -173.762,Z 1043.891,A 0.000,B 0.000,C 90.000,E1 340.315} C_DIS
LIN {X -0.069,Y -177.940,Z 1043.872,A 0.000,B 0.000,C 90.000,E1 336.922} C_DIS
LIN {X -0.008,Y -182.902,Z 1043.853,A 0.000,B 0.000,C 90.000,E1 333.512} C_DIS
LIN {X 0.103,Y -188.732,Z 1043.834,A 0.000,B 0.000,C 90.000,E1 330.127} C_DIS
LIN {X 0.060,Y -195.343,Z 1043.816,A 0.000,B 0.000,C 90.000,E1 326.834} C_DIS
LIN {X -0.098,Y -202.715,Z 1043.798,A 0.000,B 0.000,C 90.000,E1 323.623} C_DIS
LIN {X 0.136,Y -210.583,Z 1043.780,A 0.000,B 0.000,C 90.000,E1 320.356} C_DIS
LIN {X -0.004,Y -220.266,Z 1043.760,A 0.000,B 0.000,C 90.000,E1 316.863} C_DIS
LIN {X 0.003,Y -229.681,Z 1043.743,A 0.000,B 0.000,C 90.000,E1 313.785} C_DIS
LIN {X -0.023,Y -238.896,Z 1043.729,A 0.000,B 0.000,C 90.000,E1 311.148} C_DIS
LIN {X 0.039,Y -246.247,Z 1043.718,A 0.000,B 0.000,C 90.000,E1 309.277} C_DIS
LIN {X 0.049,Y -252.798,Z 1043.710,A 0.000,B 0.000,C 90.000,E1 307.810} C_DIS
LIN {X -0.044,Y -265.707,Z 1043.696,A 0.000,B 0.000,C 90.000,E1 305.311} C_DIS
LIN {X 0.126,Y -284.083,Z 1043.679,A 0.000,B 0.000,C 90.000,E1 302.133} C_DIS
LIN {X -0.027,Y -303.749,Z 1043.662,A 0.000,B 0.000,C 90.000,E1 299.127} C_DIS
LIN {X 0.081,Y -320.261,Z 1043.649,A 0.000,B 0.000,C 90.000,E1 296.821} C_DIS
LIN {X -0.111,Y -333.020,Z 1043.640,A 0.000,B 0.000,C 90.000,E1 295.283} C_DIS
LIN {X 0.062,Y -346.539,Z 1043.632,A 0.000,B 0.000,C 90.000,E1 293.770} C_DIS
LIN {X -0.145,Y -371.275,Z 1043.619,A 0.000,B 0.000,C 90.000,E1 291.408} C_DIS
LIN {X 0.217,Y -390.729,Z 1043.609,A 0.000,B 0.000,C 90.000,E1 289.631} C_DIS
LIN {X -0.066,Y -404.295,Z 1043.603,A 0.000,B 0.000,C 90.000,E1 288.489} C_DIS
LIN {X 0.089,Y -414.896,Z 1043.597,A 0.000,B 0.000,C 90.000,E1 287.511} C_DIS
LIN {X -0.193,Y -422.743,Z 1043.593,A 0.000,B 0.000,C 90.000,E1 286.804} C_DIS
LIN {X -0.144,Y -430.260,Z 1043.589,A 0.000,B 0.000,C 90.000,E1 286.024} C_DIS
LIN {X -0.085,Y -440.060,Z 1043.583,A 0.000,B 0.000,C 90.000,E1 284.954} C_DIS
LIN {X 0.231,Y -446.991,Z 1043.579,A 0.000,B 0.000,C 90.000,E1 284.120} C_DIS
LIN {X 0.061,Y -453.423,Z 1043.574,A 0.000,B 0.000,C 90.000,E1 283.355} C_DIS
LIN {X 0.223,Y -461.168,Z 1043.568,A 0.000,B 0.000,C 90.000,E1 282.299} C_DIS
LIN {X 0.182,Y -466.315,Z 1043.564,A 0.000,B 0.000,C 90.000,E1 281.535} C_DIS
LIN {X 0.089,Y -470.853,Z 1043.560,A 0.000,B 0.000,C 90.000,E1 280.782} C_DIS
LIN {X 0.126,Y -474.744,Z 1043.556,A 0.000,B 0.000,C 90.000,E1 280.018} C_DIS
LIN {X 0.110,Y -478.029,Z 1043.552,A 0.000,B 0.000,C 90.000,E1 279.265} C_DIS
LIN {X -0.223,Y -479.926,Z 1043.549,A 0.000,B 0.000,C 90.000,E1 278.803} C_DIS
LIN {X 0.157,Y -483.042,Z 1043.543,A 0.000,B 0.000,C 90.000,E1 277.757} C_DIS
LIN {X -0.152,Y -484.298,Z 1043.540,A 0.000,B 0.000,C 90.000,E1 277.296} C_DIS
LIN {X 0.029,Y -485.352,Z 1043.538,A 0.000,B 0.000,C 90.000,E1 276.777} C_DIS
LIN {X 0.219,Y -486.115,Z 1043.535,A 0.000,B 0.000,C 90.000,E1 276.258} C_DIS
LIN {X -0.071,Y -486.593,Z 1043.532,A 0.000,B 0.000,C 90.000,E1 275.796} C_DIS
LIN {X 0.128,Y -486.665,Z 1043.529,A 0.000,B 0.000,C 90.000,E1 275.277} C_DIS
LIN {X -0.197,Y -486.318,Z 1043.527,A 0.000,B 0.000,C 90.000,E1 274.821} C_DIS
LIN {X 0.005,Y -485.488,Z 1043.524,A 0.000,B 0.000,C 90.000,E1 274.302} C_DIS
LIN {X 0.201,Y -484.116,Z 1043.521,A 0.000,B 0.000,C 90.000,E1 273.784} C_DIS
LIN {X -0.122,Y -482.101,Z 1043.518,A 0.000,B 0.000,C 90.000,E1 273.326} C_DIS
LIN {X 0.222,Y -480.863,Z 1043.517,A 0.000,B 0.000,C 90.000,E1 273.037} C_DIS
LIN {X -0.113,Y -477.766,Z 1043.514,A 0.000,B 0.000,C 90.000,E1 272.579} C_DIS
LIN {X 0.015,Y -473.775,Z 1043.511,A 0.000,B 0.000,C 90.000,E1 272.064} C_DIS
LIN {X 0.136,Y -468.951,Z 1043.509,A 0.000,B 0.000,C 90.000,E1 271.547} C_DIS
LIN {X -0.077,Y -463.433,Z 1043.506,A 0.000,B 0.000,C 90.000,E1 271.088} C_DIS
LIN {X 0.032,Y -457.600,Z 1043.504,A 0.000,B 0.000,C 90.000,E1 270.630} C_DIS
LIN {X 0.053,Y -451.266,Z 1043.501,A 0.000,B 0.000,C 90.000,E1 270.229} C_DIS
LIN {X 0.049,Y -444.376,Z 1043.499,A 0.000,B 0.000,C 90.000,E1 269.885} C_DIS
LIN {X 0.153,Y -440.439,Z 1043.499,A 0.000,B 0.000,C 90.000,E1 269.714} C_DIS
LIN {X 0.026,Y -432.170,Z 1043.497,A 0.000,B 0.000,C 90.000,E1 269.484} C_DIS
LIN {X 0.041,Y -423.424,Z 1043.496,A 0.000,B 0.000,C 90.000,E1 269.312} C_DIS
LIN {X 0.053,Y -415.035,Z 1043.496,A 0.000,B 0.000,C 90.000,E1 269.198} C_DIS
LIN {X -0.017,Y -407.773,Z 1043.495,A 0.000,B 0.000,C 90.000,E1 269.141} C_DIS
LIN {X 0.123,Y -400.048,Z 1043.495,A 0.000,B 0.000,C 90.000,E1 269.083} C_DIS
LIN {X 0.020,Y -393.457,Z 1043.495,A 0.000,B 0.000,C 90.000,E1 269.083} C_DIS
LIN {X -0.014,Y -181.336,Z 1043.495,A 0.000,B 0.000,C 90.000,E1 269.083} C_DIS
LIN {X -0.001,Y -180.906,Z 1043.474,A 0.000,B 0.000,C 90.000,E1 265.355} C_DIS
LIN {X 0.072,Y -180.681,Z 1043.469,A 0.000,B 0.000,C 90.000,E1 264.489} C_DIS
LIN {X -0.029,Y -178.765,Z 1043.441,A 0.000,B 0.000,C 90.000,E1 259.454} C_DIS
LIN {X 0.043,Y -175.811,Z 1043.413,A 0.000,B 0.000,C 90.000,E1 254.338} C_DIS
LIN {X 0.037,Y -171.998,Z 1043.385,A 0.000,B 0.000,C 90.000,E1 249.209} C_DIS
LIN {X 0.012,Y -171.411,Z 1043.380,A 0.000,B 0.000,C 90.000,E1 248.358} C_DIS
LIN {X 0.059,Y -167.650,Z 1043.356,A 0.000,B 0.000,C 90.000,E1 244.024} C_DIS
LIN {X 0.073,Y -166.316,Z 1043.346,A 0.000,B 0.000,C 90.000,E1 242.281} C_DIS
LIN {X 0.067,Y -163.057,Z 1043.327,A 0.000,B 0.000,C 90.000,E1 238.791} C_DIS
LIN {X 0.029,Y -160.993,Z 1043.312,A 0.000,B 0.000,C 90.000,E1 236.167} C_DIS
LIN {X 0.006,Y -157.740,Z 1043.292,A 0.000,B 0.000,C 90.000,E1 232.637} C_DIS
LIN {X -0.056,Y -155.778,Z 1043.278,A 0.000,B 0.000,C 90.000,E1 229.989} C_DIS
LIN {X -0.001,Y -152.033,Z 1043.253,A 0.000,B 0.000,C 90.000,E1 225.486} C_DIS
LIN {X 0.017,Y -150.281,Z 1043.238,A 0.000,B 0.000,C 90.000,E1 222.771} C_DIS
LIN {X -0.056,Y -147.031,Z 1043.212,A 0.000,B 0.000,C 90.000,E1 218.257} C_DIS
LIN {X -0.064,Y -145.612,Z 1043.197,A 0.000,B 0.000,C 90.000,E1 215.518} C_DIS
LIN {X -0.064,Y -142.997,Z 1043.172,A 0.000,B 0.000,C 90.000,E1 210.924} C_DIS
LIN {X -0.007,Y -141.624,Z 1043.151,A 0.000,B 0.000,C 90.000,E1 207.206} C_DIS
LIN {X -0.082,Y -139.432,Z 1043.115,A 0.000,B 0.000,C 90.000,E1 200.737} C_DIS
LIN {X -0.027,Y -139.163,Z 1043.105,A 0.000,B 0.000,C 90.000,E1 198.852} C_DIS
LIN {X 0.010,Y -138.340,Z 1043.058,A 0.000,B 0.000,C 90.000,E1 190.433} C_DIS
LIN {X 0.017,Y -139.477,Z 1043.006,A 0.000,B 0.000,C 90.000,E1 181.088} C_DIS
LIN {X -0.042,Y -141.062,Z 1042.975,A 0.000,B 0.000,C 90.000,E1 175.527} C_DIS
LIN {X 0.053,Y -142.435,Z 1042.960,A 0.000,B 0.000,C 90.000,E1 172.704} C_DIS
LIN {X -0.028,Y -144.674,Z 1042.934,A 0.000,B 0.000,C 90.000,E1 168.117} C_DIS
LIN {X -0.045,Y -147.261,Z 1042.913,A 0.000,B 0.000,C 90.000,E1 164.448} C_DIS
LIN {X -0.027,Y -150.579,Z 1042.888,A 0.000,B 0.000,C 90.000,E1 159.880} C_DIS
LIN {X 0.052,Y -154.050,Z 1042.868,A 0.000,B 0.000,C 90.000,E1 156.230} C_DIS
LIN {X -0.021,Y -157.467,Z 1042.848,A 0.000,B 0.000,C 90.000,E1 152.666} C_DIS
LIN {X 0.066,Y -161.689,Z 1042.828,A 0.000,B 0.000,C 90.000,E1 149.076} C_DIS
LIN {X -0.057,Y -165.883,Z 1042.809,A 0.000,B 0.000,C 90.000,E1 145.595} C_DIS
LIN {X -0.067,Y -170.863,Z 1042.789,A 0.000,B 0.000,C 90.000,E1 142.110} C_DIS
LIN {X -0.020,Y -175.733,Z 1042.770,A 0.000,B 0.000,C 90.000,E1 138.647} C_DIS
LIN {X -0.030,Y -181.343,Z 1042.751,A 0.000,B 0.000,C 90.000,E1 135.243} C_DIS
LIN {X 0.104,Y -186.833,Z 1042.733,A 0.000,B 0.000,C 90.000,E1 131.838} C_DIS
LIN {X 0.058,Y -191.420,Z 1042.719,A 0.000,B 0.000,C 90.000,E1 129.358} C_DIS
LIN {X -0.073,Y -197.708,Z 1042.699,A 0.000,B 0.000,C 90.000,E1 125.884} C_DIS
LIN {X -0.020,Y -197.743,Z 1042.699,A 0.000,B 0.000,C 90.000,E1 125.851} C_DIS
LIN {X 0.167,Y -302.916,Z 1042.699,A 0.000,B 0.000,C 90.000,E1 125.804} C_DIS
LIN {X 0.119,Y -304.058,Z 1042.699,A 0.000,B 0.000,C 90.000,E1 125.804} C_DIS
LIN {X 0.056,Y -308.242,Z 1042.698,A 0.000,B 0.000,C 90.000,E1 125.678} C_DIS
LIN {X 0.173,Y -310.386,Z 1042.698,A 0.000,B 0.000,C 90.000,E1 125.518} C_DIS
LIN {X 0.046,Y -313.332,Z 1042.696,A 0.000,B 0.000,C 90.000,E1 125.264} C_DIS
LIN {X -0.006,Y -317.021,Z 1042.693,A 0.000,B 0.000,C 90.000,E1 124.739} C_DIS
LIN {X 0.051,Y -318.580,Z 1042.691,A 0.000,B 0.000,C 90.000,E1 124.405} C_DIS
LIN {X -0.004,Y -321.928,Z 1042.686,A 0.000,B 0.000,C 90.000,E1 123.452} C_DIS
LIN {X 0.059,Y -332.247,Z 1042.670,A 0.000,B 0.000,C 90.000,E1 120.590} C_DIS
LIN {X 0.193,Y -343.909,Z 1042.654,A 0.000,B 0.000,C 90.000,E1 117.769} C_DIS
LIN {X -0.126,Y -357.011,Z 1042.639,A 0.000,B 0.000,C 90.000,E1 115.079} C_DIS
LIN {X 0.190,Y -369.963,Z 1042.626,A 0.000,B 0.000,C 90.000,E1 112.642} C_DIS
LIN {X 0.220,Y -384.237,Z 1042.613,A 0.000,B 0.000,C 90.000,E1 110.301} C_DIS
LIN {X -0.030,Y -399.934,Z 1042.600,A 0.000,B 0.000,C 90.000,E1 108.055} C_DIS
LIN {X -0.151,Y -417.166,Z 1042.588,A 0.000,B 0.000,C 90.000,E1 105.843} C_DIS
LIN {X 0.043,Y -436.051,Z 1042.576,A 0.000,B 0.000,C 90.000,E1 103.647} C_DIS
LIN {X 0.131,Y -456.074,Z 1042.564,A 0.000,B 0.000,C 90.000,E1 101.591} C_DIS
LIN {X -0.082,Y -466.296,Z 1042.559,A 0.000,B 0.000,C 90.000,E1 100.658} C_DIS
LIN {X -0.073,Y -468.628,Z 1042.558,A 0.000,B 0.000,C 90.000,E1 100.423} C_DIS
LIN {X 0.198,Y -470.477,Z 1042.557,A 0.000,B 0.000,C 90.000,E1 100.141} C_DIS
LIN {X 0.092,Y -471.872,Z 1042.555,A 0.000,B 0.000,C 90.000,E1 99.905} C_DIS
LIN {X -0.198,Y -473.690,Z 1042.552,A 0.000,B 0.000,C 90.000,E1 99.434} C_DIS
LIN {X -0.090,Y -474.416,Z 1042.549,A 0.000,B 0.000,C 90.000,E1 98.916} C_DIS
LIN {X 0.031,Y -474.171,Z 1042.547,A 0.000,B 0.000,C 90.000,E1 98.398} C_DIS
LIN {X 0.224,Y -472.927,Z 1042.544,A 0.000,B 0.000,C 90.000,E1 97.871} C_DIS
LIN {X 0.020,Y -471.871,Z 1042.542,A 0.000,B 0.000,C 90.000,E1 97.644} C_DIS
LIN {X -0.119,Y -470.455,Z 1042.541,A 0.000,B 0.000,C 90.000,E1 97.409} C_DIS
LIN {X -0.069,Y -458.046,Z 1042.531,A 0.000,B 0.000,C 90.000,E1 95.625} C_DIS
LIN {X -0.065,Y -443.753,Z 1042.520,A 0.000,B 0.000,C 90.000,E1 93.555} C_DIS
LIN {X 0.167,Y -428.889,Z 1042.506,A 0.000,B 0.000,C 90.000,E1 91.146} C_DIS
LIN {X -0.111,Y -416.566,Z 1042.495,A 0.000,B 0.000,C 90.000,E1 89.026} C_DIS
LIN {X 0.025,Y -407.882,Z 1042.485,A 0.000,B 0.000,C 90.000,E1 87.364} C_DIS
LIN {X 0.026,Y -398.969,Z 1042.476,A 0.000,B 0.000,C 90.000,E1 85.698} C_DIS
LIN {X -0.132,Y -389.844,Z 1042.467,A 0.000,B 0.000,C 90.000,E1 84.033} C_DIS
LIN {X 0.013,Y -380.537,Z 1042.457,A 0.000,B 0.000,C 90.000,E1 82.299} C_DIS
LIN {X 0.040,Y -372.554,Z 1042.449,A 0.000,B 0.000,C 90.000,E1 80.849} C_DIS
LIN {X -0.091,Y -361.003,Z 1042.438,A 0.000,B 0.000,C 90.000,E1 78.814} C_DIS
LIN {X 0.021,Y -349.359,Z 1042.426,A 0.000,B 0.000,C 90.000,E1 76.700} C_DIS
LIN {X -0.030,Y -337.857,Z 1042.414,A 0.000,B 0.000,C 90.000,E1 74.574} C_DIS
LIN {X -0.012,Y -323.602,Z 1042.399,A 0.000,B 0.000,C 90.000,E1 71.764} C_DIS
LIN {X 0.002,Y -311.347,Z 1042.385,A 0.000,B 0.000,C 90.000,E1 69.209} C_DIS
LIN {X -0.058,Y -299.583,Z 1042.370,A 0.000,B 0.000,C 90.000,E1 66.613} C_DIS
LIN {X -0.042,Y -288.069,Z 1042.355,A 0.000,B 0.000,C 90.000,E1 63.948} C_DIS
LIN {X 0.000,Y -278.214,Z 1042.342,A 0.000,B 0.000,C 90.000,E1 61.563} C_DIS
LIN {X 0.015,Y -267.180,Z 1042.327,A 0.000,B 0.000,C 90.000,E1 58.791} C_DIS
LIN {X 0.125,Y -257.743,Z 1042.313,A 0.000,B 0.000,C 90.000,E1 56.294} C_DIS
LIN {X 0.106,Y -247.255,Z 1042.297,A 0.000,B 0.000,C 90.000,E1 53.417} C_DIS
LIN {X 0.066,Y -236.106,Z 1042.278,A 0.000,B 0.000,C 90.000,E1 50.114} C_DIS
LIN {X -0.001,Y -225.704,Z 1042.260,A 0.000,B 0.000,C 90.000,E1 46.743} C_DIS
LIN {X 0.134,Y -218.145,Z 1042.245,A 0.000,B 0.000,C 90.000,E1 44.028} C_DIS
LIN {X 0.025,Y -209.943,Z 1042.228,A 0.000,B 0.000,C 90.000,E1 40.943} C_DIS
LIN {X -0.095,Y -202.237,Z 1042.210,A 0.000,B 0.000,C 90.000,E1 37.810} C_DIS
LIN {X 0.102,Y -195.057,Z 1042.192,A 0.000,B 0.000,C 90.000,E1 34.532} C_DIS
LIN {X 0.104,Y -188.543,Z 1042.174,A 0.000,B 0.000,C 90.000,E1 31.258} C_DIS
LIN {X -0.012,Y -182.787,Z 1042.155,A 0.000,B 0.000,C 90.000,E1 27.975} C_DIS
LIN {X 0.055,Y -177.772,Z 1042.137,A 0.000,B 0.000,C 90.000,E1 24.591} C_DIS
LIN {X -0.056,Y -173.538,Z 1042.118,A 0.000,B 0.000,C 90.000,E1 21.227} C_DIS
LIN {X 0.031,Y -169.998,Z 1042.099,A 0.000,B 0.000,C 90.000,E1 17.764} C_DIS
LIN {X 0.097,Y -166.606,Z 1042.075,A 0.000,B 0.000,C 90.000,E1 13.411} C_DIS
LIN {X -0.040,Y -163.964,Z 1042.046,A 0.000,B 0.000,C 90.000,E1 8.219} C_DIS
LIN {X 0.057,Y -164.838,Z 1041.953,A 0.000,B 0.000,C 90.000,E1 351.602} C_DIS
LIN {X 0.063,Y -167.344,Z 1041.929,A 0.000,B 0.000,C 90.000,E1 347.229} C_DIS
LIN {X 0.004,Y -171.011,Z 1041.905,A 0.000,B 0.000,C 90.000,E1 342.906} C_DIS
LIN {X 0.050,Y -174.654,Z 1041.886,A 0.000,B 0.000,C 90.000,E1 339.444} C_DIS
LIN {X -0.018,Y -178.993,Z 1041.867,A 0.000,B 0.000,C 90.000,E1 336.049} C_DIS
LIN {X -0.013,Y -184.193,Z 1041.848,A 0.000,B 0.000,C 90.000,E1 332.666} C_DIS
LIN {X -0.034,Y -190.242,Z 1041.830,A 0.000,B 0.000,C 90.000,E1 329.331} C_DIS
LIN {X 0.063,Y -197.079,Z 1041.811,A 0.000,B 0.000,C 90.000,E1 326.008} C_DIS
LIN {X 0.066,Y -204.583,Z 1041.793,A 0.000,B 0.000,C 90.000,E1 322.763} C_DIS
LIN {X 0.034,Y -212.619,Z 1041.776,A 0.000,B 0.000,C 90.000,E1 319.585} C_DIS
LIN {X 0.102,Y -222.467,Z 1041.756,A 0.000,B 0.000,C 90.000,E1 316.053} C_DIS
LIN {X 0.013,Y -232.124,Z 1041.739,A 0.000,B 0.000,C 90.000,E1 313.014} C_DIS
LIN {X -0.087,Y -240.218,Z 1041.726,A 0.000,B 0.000,C 90.000,E1 310.782} C_DIS
LIN {X -0.007,Y -247.742,Z 1041.716,A 0.000,B 0.000,C 90.000,E1 308.910} C_DIS
LIN {X 0.020,Y -254.488,Z 1041.708,A 0.000,B 0.000,C 90.000,E1 307.443} C_DIS
LIN {X -0.088,Y -265.664,Z 1041.696,A 0.000,B 0.000,C 90.000,E1 305.311} C_DIS
LIN {X 0.077,Y -284.033,Z 1041.679,A 0.000,B 0.000,C 90.000,E1 302.133} C_DIS
LIN {X -0.081,Y -303.776,Z 1041.662,A 0.000,B 0.000,C 90.000,E1 299.127} C_DIS
LIN {X 0.026,Y -320.351,Z 1041.649,A 0.000,B 0.000,C 90.000,E1 296.821} C_DIS
LIN {X -0.166,Y -333.177,Z 1041.640,A 0.000,B 0.000,C 90.000,E1 295.283} C_DIS
LIN {X -0.119,Y -346.440,Z 1041.632,A 0.000,B 0.000,C 90.000,E1 293.823} C_DIS
LIN {X 0.066,Y -371.051,Z 1041.619,A 0.000,B 0.000,C 90.000,E1 291.408} C_DIS
LIN {X 0.050,Y -387.563,Z 1041.611,A 0.000,B 0.000,C 90.000,E1 289.939} C_DIS
LIN {X -0.130,Y -401.165,Z 1041.604,A 0.000,B 0.000,C 90.000,E1 288.779} C_DIS
LIN {X -0.095,Y -411.885,Z 1041.599,A 0.000,B 0.000,C 90.000,E1 287.819} C_DIS
LIN {X -0.144,Y -419.722,Z 1041.595,A 0.000,B 0.000,C 90.000,E1 287.094} C_DIS
LIN {X 0.010,Y -427.278,Z 1041.591,A 0.000,B 0.000,C 90.000,E1 286.315} C_DIS
LIN {X -0.136,Y -434.653,Z 1041.586,A 0.000,B 0.000,C 90.000,E1 285.552} C_DIS
LIN {X -0.091,Y -444.220,Z 1041.580,A 0.000,B 0.000,C 90.000,E1 284.481} C_DIS
LIN {X -0.174,Y -450.870,Z 1041.576,A 0.000,B 0.000,C 90.000,E1 283.703} C_DIS
LIN {X 0.127,Y -456.919,Z 1041.572,A 0.000,B 0.000,C 90.000,E1 282.883} C_DIS
LIN {X -0.123,Y -464.277,Z 1041.566,A 0.000,B 0.000,C 90.000,E1 281.883} C_DIS
LIN {X -0.236,Y -469.039,Z 1041.562,A 0.000,B 0.000,C 90.000,E1 281.130} C_DIS
LIN {X 0.246,Y -473.227,Z 1041.557,A 0.000,B 0.000,C 90.000,E1 280.310} C_DIS
LIN {X 0.222,Y -476.787,Z 1041.553,A 0.000,B 0.000,C 90.000,E1 279.557} C_DIS
LIN {X -0.247,Y -479.773,Z 1041.549,A 0.000,B 0.000,C 90.000,E1 278.859} C_DIS
LIN {X -0.101,Y -481.475,Z 1041.546,A 0.000,B 0.000,C 90.000,E1 278.341} C_DIS
LIN {X 0.127,Y -482.962,Z 1041.543,A 0.000,B 0.000,C 90.000,E1 277.814} C_DIS
LIN {X -0.002,Y -485.317,Z 1041.538,A 0.000,B 0.000,C 90.000,E1 276.834} C_DIS
LIN {X 0.186,Y -486.122,Z 1041.535,A 0.000,B 0.000,C 90.000,E1 276.315} C_DIS
LIN {X -0.102,Y -486.643,Z 1041.532,A 0.000,B 0.000,C 90.000,E1 275.853} C_DIS
LIN {X 0.095,Y -486.764,Z 1041.530,A 0.000,B 0.000,C 90.000,E1 275.334} C_DIS
LIN {X -0.230,Y -486.504,Z 1041.527,A 0.000,B 0.000,C 90.000,E1 274.878} C_DIS
LIN {X -0.028,Y -485.726,Z 1041.524,A 0.000,B 0.000,C 90.000,E1 274.359} C_DIS
LIN {X 0.169,Y -484.417,Z 1041.521,A 0.000,B 0.000,C 90.000,E1 273.841} C_DIS
LIN {X -0.152,Y -482.506,Z 1041.519,A 0.000,B 0.000,C 90.000,E1 273.383} C_DIS
LIN {X 0.192,Y -481.311,Z 1041.517,A 0.000,B 0.000,C 90.000,E1 273.094} C_DIS
LIN {X -0.142,Y -478.311,Z 1041.515,A 0.000,B 0.000,C 90.000,E1 272.636} C_DIS
LIN {X -0.010,Y -474.456,Z 1041.512,A 0.000,B 0.000,C 90.000,E1 272.121} C_DIS
LIN {X 0.115,Y -469.766,Z 1041.509,A 0.000,B 0.000,C 90.000,E1 271.604} C_DIS
LIN {X -0.144,Y -464.340,Z 1041.506,A 0.000,B 0.000,C 90.000,E1 271.146} C_DIS
LIN {X -0.111,Y -458.484,Z 1041.504,A 0.000,B 0.000,C 90.000,E1 270.688} C_DIS
LIN {X -0.166,Y -452.161,Z 1041.501,A 0.000,B 0.000,C 90.000,E1 270.286} C_DIS
LIN {X 0.128,Y -448.695,Z 1041.500,A 0.000,B 0.000,C 90.000,E1 270.057} C_DIS
LIN {X -0.169,Y -441.356,Z 1041.499,A 0.000,B 0.000,C 90.000,E1 269.771} C_DIS
LIN {X 0.183,Y -437.735,Z 1041.498,A 0.000,B 0.000,C 90.000,E1 269.599} C_DIS
LIN {X -0.128,Y -429.497,Z 1041.497,A 0.000,B 0.000,C 90.000,E1 269.427} C_DIS
LIN {X 0.075,Y -420.766,Z 1041.496,A 0.000,B 0.000,C 90.000,E1 269.255} C_DIS
LIN {X 0.152,Y -412.263,Z 1041.495,A 0.000,B 0.000,C 90.000,E1 269.141} C_DIS
LIN {X 0.111,Y -402.846,Z 1041.495,A 0.000,B 0.000,C 90.000,E1 269.083} C_DIS
LIN {X -0.064,Y -392.872,Z 1041.495,A 0.000,B 0.000,C 90.000,E1 269.083} C_DIS
LIN {X -0.056,Y -181.333,Z 1041.495,A 0.000,B 0.000,C 90.000,E1 269.083} C_DIS
LIN {X -0.025,Y -180.905,Z 1041.474,A 0.000,B 0.000,C 90.000,E1 265.355} C_DIS
LIN {X 0.048,Y -180.678,Z 1041.469,A 0.000,B 0.000,C 90.000,E1 264.489} C_DIS
LIN {X -0.053,Y -178.760,Z 1041.441,A 0.000,B 0.000,C 90.000,E1 259.454} C_DIS
LIN {X 0.019,Y -175.807,Z 1041.413,A 0.000,B 0.000,C 90.000,E1 254.338} C_DIS
LIN {X 0.014,Y -171.993,Z 1041.385,A 0.000,B 0.000,C 90.000,E1 249.209} C_DIS
LIN {X 0.052,Y -171.404,Z 1041.380,A 0.000,B 0.000,C 90.000,E1 248.337} C_DIS
LIN {X 0.036,Y -167.645,Z 1041.356,A 0.000,B 0.000,C 90.000,E1 244.024} C_DIS
LIN {X 0.051,Y -166.307,Z 1041.346,A 0.000,B 0.000,C 90.000,E1 242.281} C_DIS
LIN {X 0.044,Y -163.051,Z 1041.327,A 0.000,B 0.000,C 90.000,E1 238.791} C_DIS
LIN {X 0.006,Y -160.984,Z 1041.312,A 0.000,B 0.000,C 90.000,E1 236.167} C_DIS
LIN {X -0.017,Y -157.733,Z 1041.292,A 0.000,B 0.000,C 90.000,E1 232.637} C_DIS
LIN {X -0.078,Y -155.772,Z 1041.278,A 0.000,B 0.000,C 90.000,E1 229.989} C_DIS
LIN {X -0.022,Y -152.027,Z 1041.253,A 0.000,B 0.000,C 90.000,E1 225.486} C_DIS
LIN {X -0.004,Y -150.275,Z 1041.238,A 0.000,B 0.000,C 90.000,E1 222.771} C_DIS
LIN {X 0.013,Y -147.026,Z 1041.212,A 0.000,B 0.000,C 90.000,E1 218.222} C_DIS
LIN {X 0.033,Y -145.608,Z 1041.197,A 0.000,B 0.000,C 90.000,E1 215.471} C_DIS
LIN {X 0.037,Y -142.993,Z 1041.172,A 0.000,B 0.000,C 90.000,E1 210.875} C_DIS
LIN {X -0.027,Y -141.620,Z 1041.151,A 0.000,B 0.000,C 90.000,E1 207.206} C_DIS
LIN {X 0.029,Y -139.431,Z 1041.115,A 0.000,B 0.000,C 90.000,E1 200.684} C_DIS
LIN {X -0.048,Y -139.162,Z 1041.105,A 0.000,B 0.000,C 90.000,E1 198.852} C_DIS
LIN {X -0.011,Y -138.341,Z 1041.058,A 0.000,B 0.000,C 90.000,E1 190.433} C_DIS
LIN {X -0.003,Y -139.479,Z 1041.006,A 0.000,B 0.000,C 90.000,E1 181.088} C_DIS
LIN {X -0.063,Y -141.066,Z 1040.975,A 0.000,B 0.000,C 90.000,E1 175.527} C_DIS
LIN {X 0.032,Y -142.440,Z 1040.960,A 0.000,B 0.000,C 90.000,E1 172.704} C_DIS
LIN {X -0.048,Y -144.678,Z 1040.934,A 0.000,B 0.000,C 90.000,E1 168.117} C_DIS
LIN {X 0.076,Y -147.268,Z 1040.913,A 0.000,B 0.000,C 90.000,E1 164.393} C_DIS
LIN {X -0.049,Y -150.586,Z 1040.888,A 0.000,B 0.000,C 90.000,E1 159.880} C_DIS
LIN {X 0.030,Y -154.057,Z 1040.868,A 0.000,B 0.000,C 90.000,E1 156.230} C_DIS
LIN {X -0.043,Y -157.476,Z 1040.848,A 0.000,B 0.000,C 90.000,E1 152.666} C_DIS
LIN {X 0.043,Y -161.699,Z 1040.828,A 0.000,B 0.000,C 90.000,E1 149.076} C_DIS
LIN {X -0.080,Y -165.893,Z 1040.809,A 0.000,B 0.000,C 90.000,E1 145.595} C_DIS
LIN {X 0.045,Y -170.876,Z 1040.789,A 0.000,B 0.000,C 90.000,E1 142.065} C_DIS
LIN {X 0.072,Y -175.744,Z 1040.770,A 0.000,B 0.000,C 90.000,E1 138.609} C_DIS
LIN {X -0.054,Y -181.354,Z 1040.751,A 0.000,B 0.000,C 90.000,E1 135.243} C_DIS
LIN {X 0.080,Y -186.846,Z 1040.733,A 0.000,B 0.000,C 90.000,E1 131.838} C_DIS
LIN {X 0.033,Y -191.432,Z 1040.719,A 0.000,B 0.000,C 90.000,E1 129.358} C_DIS
LIN {X -0.004,Y -197.669,Z 1040.699,A 0.000,B 0.000,C 90.000,E1 125.884} C_DIS
LIN {X -0.042,Y -303.157,Z 1040.699,A 0.000,B 0.000,C 90.000,E1 125.884} C_DIS
LIN {X 0.082,Y -306.037,Z 1040.699,A 0.000,B 0.000,C 90.000,E1 125.804} C_DIS
LIN {X 0.135,Y -310.853,Z 1040.698,A 0.000,B 0.000,C 90.000,E1 125.518} C_DIS
LIN {X 0.006,Y -313.600,Z 1040.696,A 0.000,B 0.000,C 90.000,E1 125.264} C_DIS
LIN {X 0.047,Y -317.281,Z 1040.693,A 0.000,B 0.000,C 90.000,E1 124.692} C_DIS
LIN {X -0.157,Y -318.750,Z 1040.691,A 0.000,B 0.000,C 90.000,E1 124.405} C_DIS
LIN {X -0.151,Y -332.367,Z 1040.670,A 0.000,B 0.000,C 90.000,E1 120.590} C_DIS
LIN {X -0.022,Y -344.046,Z 1040.654,A 0.000,B 0.000,C 90.000,E1 117.769} C_DIS
LIN {X -0.022,Y -357.168,Z 1040.639,A 0.000,B 0.000,C 90.000,E1 115.027} C_DIS
LIN {X -0.032,Y -370.137,Z 1040.626,A 0.000,B 0.000,C 90.000,E1 112.642} C_DIS
LIN {X -0.006,Y -384.430,Z 1040.613,A 0.000,B 0.000,C 90.000,E1 110.301} C_DIS
LIN {X 0.120,Y -400.149,Z 1040.600,A 0.000,B 0.000,C 90.000,E1 108.000} C_DIS
LIN {X 0.014,Y -417.404,Z 1040.588,A 0.000,B 0.000,C 90.000,E1 105.788} C_DIS
LIN {X -0.196,Y -436.312,Z 1040.576,A 0.000,B 0.000,C 90.000,E1 103.647} C_DIS
LIN {X -0.099,Y -456.343,Z 1040.564,A 0.000,B 0.000,C 90.000,E1 101.591} C_DIS
LIN {X 0.152,Y -466.570,Z 1040.559,A 0.000,B 0.000,C 90.000,E1 100.602} C_DIS
LIN {X 0.164,Y -468.832,Z 1040.558,A 0.000,B 0.000,C 90.000,E1 100.366} C_DIS
LIN {X -0.062,Y -470.653,Z 1040.556,A 0.000,B 0.000,C 90.000,E1 100.141} C_DIS
LIN {X -0.205,Y -472.022,Z 1040.555,A 0.000,B 0.000,C 90.000,E1 99.905} C_DIS
LIN {X -0.026,Y -473.756,Z 1040.552,A 0.000,B 0.000,C 90.000,E1 99.378} C_DIS
LIN {X 0.083,Y -474.413,Z 1040.549,A 0.000,B 0.000,C 90.000,E1 98.859} C_DIS
LIN {X 0.206,Y -474.104,Z 1040.547,A 0.000,B 0.000,C 90.000,E1 98.341} C_DIS
LIN {X -0.070,Y -472.787,Z 1040.544,A 0.000,B 0.000,C 90.000,E1 97.871} C_DIS
LIN {X 0.195,Y -471.685,Z 1040.542,A 0.000,B 0.000,C 90.000,E1 97.587} C_DIS
LIN {X 0.055,Y -470.214,Z 1040.541,A 0.000,B 0.000,C 90.000,E1 97.352} C_DIS
LIN {X 0.097,Y -457.809,Z 1040.531,A 0.000,B 0.000,C 90.000,E1 95.568} C_DIS
LIN {X 0.092,Y -443.515,Z 1040.520,A 0.000,B 0.000,C 90.000,E1 93.498} C_DIS
LIN {X -0.115,Y -428.655,Z 1040.506,A 0.000,B 0.000,C 90.000,E1 91.146} C_DIS
LIN {X 0.025,Y -416.369,Z 1040.494,A 0.000,B 0.000,C 90.000,E1 88.969} C_DIS
LIN {X -0.182,Y -406.202,Z 1040.484,A 0.000,B 0.000,C 90.000,E1 87.078} C_DIS
LIN {X -0.139,Y -395.755,Z 1040.473,A 0.000,B 0.000,C 90.000,E1 85.122} C_DIS
LIN {X 0.077,Y -386.553,Z 1040.463,A 0.000,B 0.000,C 90.000,E1 83.394} C_DIS
LIN {X 0.166,Y -377.177,Z 1040.454,A 0.000,B 0.000,C 90.000,E1 81.659} C_DIS
LIN {X 0.142,Y -369.040,Z 1040.446,A 0.000,B 0.000,C 90.000,E1 80.208} C_DIS
LIN {X -0.033,Y -359.104,Z 1040.436,A 0.000,B 0.000,C 90.000,E1 78.465} C_DIS
LIN {X 0.038,Y -347.507,Z 1040.424,A 0.000,B 0.000,C 90.000,E1 76.353} C_DIS
LIN {X -0.076,Y -334.429,Z 1040.411,A 0.000,B 0.000,C 90.000,E1 73.921} C_DIS
LIN {X 0.001,Y -321.880,Z 1040.397,A 0.000,B 0.000,C 90.000,E1 71.402} C_DIS
LIN {X -0.085,Y -306.737,Z 1040.379,A 0.000,B 0.000,C 90.000,E1 68.209} C_DIS
LIN {X 0.141,Y -295.042,Z 1040.364,A 0.000,B 0.000,C 90.000,E1 65.537} C_DIS
LIN {X 0.041,Y -283.644,Z 1040.349,A 0.000,B 0.000,C 90.000,E1 62.871} C_DIS
LIN {X 0.104,Y -273.852,Z 1040.336,A 0.000,B 0.000,C 90.000,E1 60.461} C_DIS
LIN {X -0.086,Y -262.918,Z 1040.321,A 0.000,B 0.000,C 90.000,E1 57.709} C_DIS
LIN {X -0.043,Y -252.232,Z 1040.305,A 0.000,B 0.000,C 90.000,E1 54.848} C_DIS
LIN {X 0.093,Y -240.735,Z 1040.286,A 0.000,B 0.000,C 90.000,E1 51.537} C_DIS
LIN {X -0.156,Y -230.031,Z 1040.268,A 0.000,B 0.000,C 90.000,E1 48.243} C_DIS
LIN {X 0.080,Y -220.072,Z 1040.249,A 0.000,B 0.000,C 90.000,E1 44.757} C_DIS
LIN {X 0.004,Y -211.722,Z 1040.232,A 0.000,B 0.000,C 90.000,E1 41.676} C_DIS
LIN {X -0.077,Y -203.892,Z 1040.214,A 0.000,B 0.000,C 90.000,E1 38.543} C_DIS
LIN {X 0.005,Y -196.575,Z 1040.196,A 0.000,B 0.000,C 90.000,E1 35.311} C_DIS
LIN {X -0.007,Y -189.867,Z 1040.178,A 0.000,B 0.000,C 90.000,E1 32.054} C_DIS
LIN {X -0.001,Y -183.922,Z 1040.160,A 0.000,B 0.000,C 90.000,E1 28.743} C_DIS
LIN {X -0.071,Y -178.725,Z 1040.141,A 0.000,B 0.000,C 90.000,E1 25.412} C_DIS
LIN {X -0.089,Y -174.332,Z 1040.122,A 0.000,B 0.000,C 90.000,E1 22.025} C_DIS
LIN {X 0.073,Y -170.623,Z 1040.103,A 0.000,B 0.000,C 90.000,E1 18.544} C_DIS
LIN {X -0.003,Y -167.049,Z 1040.079,A 0.000,B 0.000,C 90.000,E1 14.245} C_DIS
LIN {X -0.056,Y -164.177,Z 1040.050,A 0.000,B 0.000,C 90.000,E1 9.029} C_DIS
LIN {X -0.030,Y -162.563,Z 1039.997,A 0.000,B 0.000,C 90.000,E1 359.542} C_DIS
LIN {X 0.079,Y -164.353,Z 1039.958,A 0.000,B 0.000,C 90.000,E1 352.470} C_DIS
LIN {X 0.055,Y -167.270,Z 1039.929,A 0.000,B 0.000,C 90.000,E1 347.229} C_DIS
LIN {X -0.006,Y -170.929,Z 1039.905,A 0.000,B 0.000,C 90.000,E1 342.906} C_DIS
LIN {X 0.037,Y -174.561,Z 1039.886,A 0.000,B 0.000,C 90.000,E1 339.444} C_DIS
LIN {X -0.033,Y -178.913,Z 1039.867,A 0.000,B 0.000,C 90.000,E1 336.049} C_DIS
LIN {X -0.032,Y -184.114,Z 1039.848,A 0.000,B 0.000,C 90.000,E1 332.666} C_DIS
LIN {X -0.055,Y -190.179,Z 1039.829,A 0.000,B 0.000,C 90.000,E1 329.331} C_DIS
LIN {X 0.040,Y -197.036,Z 1039.811,A 0.000,B 0.000,C 90.000,E1 326.008} C_DIS
LIN {X 0.042,Y -204.527,Z 1039.793,A 0.000,B 0.000,C 90.000,E1 322.763} C_DIS
LIN {X 0.007,Y -212.585,Z 1039.776,A 0.000,B 0.000,C 90.000,E1 319.585} C_DIS
LIN {X 0.073,Y -222.402,Z 1039.756,A 0.000,B 0.000,C 90.000,E1 316.053} C_DIS
LIN {X -0.019,Y -232.053,Z 1039.739,A 0.000,B 0.000,C 90.000,E1 313.014} C_DIS
LIN {X 0.035,Y -240.121,Z 1039.726,A 0.000,B 0.000,C 90.000,E1 310.744} C_DIS
LIN {X -0.045,Y -247.673,Z 1039.716,A 0.000,B 0.000,C 90.000,E1 308.910} C_DIS
LIN {X -0.019,Y -254.411,Z 1039.708,A 0.000,B 0.000,C 90.000,E1 307.443} C_DIS
LIN {X -0.131,Y -265.614,Z 1039.696,A 0.000,B 0.000,C 90.000,E1 305.311} C_DIS
LIN {X 0.030,Y -283.988,Z 1039.679,A 0.000,B 0.000,C 90.000,E1 302.133} C_DIS
LIN {X 0.134,Y -303.825,Z 1039.662,A 0.000,B 0.000,C 90.000,E1 299.077} C_DIS
LIN {X -0.026,Y -320.449,Z 1039.649,A 0.000,B 0.000,C 90.000,E1 296.821} C_DIS
LIN {X 0.123,Y -333.481,Z 1039.640,A 0.000,B 0.000,C 90.000,E1 295.207} C_DIS
LIN {X -0.045,Y -346.935,Z 1039.632,A 0.000,B 0.000,C 90.000,E1 293.770} C_DIS
LIN {X 0.115,Y -374.512,Z 1039.617,A 0.000,B 0.000,C 90.000,E1 291.099} C_DIS
LIN {X 0.219,Y -390.931,Z 1039.609,A 0.000,B 0.000,C 90.000,E1 289.631} C_DIS
LIN {X -0.129,Y -404.517,Z 1039.603,A 0.000,B 0.000,C 90.000,E1 288.489} C_DIS
LIN {X -0.030,Y -415.175,Z 1039.597,A 0.000,B 0.000,C 90.000,E1 287.511} C_DIS
LIN {X -0.260,Y -422.852,Z 1039.593,A 0.000,B 0.000,C 90.000,E1 286.804} C_DIS
LIN {X 0.077,Y -432.738,Z 1039.587,A 0.000,B 0.000,C 90.000,E1 285.733} C_DIS
LIN {X 0.158,Y -442.318,Z 1039.582,A 0.000,B 0.000,C 90.000,E1 284.662} C_DIS
LIN {X 0.058,Y -449.128,Z 1039.577,A 0.000,B 0.000,C 90.000,E1 283.883} C_DIS
LIN {X -0.089,Y -455.309,Z 1039.573,A 0.000,B 0.000,C 90.000,E1 283.119} C_DIS
LIN {X 0.092,Y -462.842,Z 1039.567,A 0.000,B 0.000,C 90.000,E1 282.063} C_DIS
LIN {X 0.057,Y -467.783,Z 1039.563,A 0.000,B 0.000,C 90.000,E1 281.299} C_DIS
LIN {X -0.020,Y -472.134,Z 1039.559,A 0.000,B 0.000,C 90.000,E1 280.546} C_DIS
LIN {X -0.059,Y -475.885,Z 1039.554,A 0.000,B 0.000,C 90.000,E1 279.792} C_DIS
LIN {X 0.145,Y -478.075,Z 1039.552,A 0.000,B 0.000,C 90.000,E1 279.265} C_DIS
LIN {X -0.187,Y -479.992,Z 1039.549,A 0.000,B 0.000,C 90.000,E1 278.803} C_DIS
LIN {X 0.032,Y -481.682,Z 1039.546,A 0.000,B 0.000,C 90.000,E1 278.276} C_DIS
LIN {X 0.193,Y -483.140,Z 1039.543,A 0.000,B 0.000,C 90.000,E1 277.757} C_DIS
LIN {X -0.115,Y -484.405,Z 1039.540,A 0.000,B 0.000,C 90.000,E1 277.296} C_DIS
LIN {X 0.066,Y -485.461,Z 1039.538,A 0.000,B 0.000,C 90.000,E1 276.777} C_DIS
LIN {X -0.227,Y -486.217,Z 1039.535,A 0.000,B 0.000,C 90.000,E1 276.315} C_DIS
LIN {X -0.032,Y -486.712,Z 1039.532,A 0.000,B 0.000,C 90.000,E1 275.796} C_DIS
LIN {X 0.168,Y -486.853,Z 1039.529,A 0.000,B 0.000,C 90.000,E1 275.277} C_DIS
LIN {X -0.158,Y -486.562,Z 1039.527,A 0.000,B 0.000,C 90.000,E1 274.821} C_DIS
LIN {X 0.046,Y -485.770,Z 1039.524,A 0.000,B 0.000,C 90.000,E1 274.302} C_DIS
LIN {X 0.243,Y -484.409,Z 1039.521,A 0.000,B 0.000,C 90.000,E1 273.784} C_DIS
LIN {X -0.078,Y -482.481,Z 1039.518,A 0.000,B 0.000,C 90.000,E1 273.326} C_DIS
LIN {X 0.103,Y -479.790,Z 1039.516,A 0.000,B 0.000,C 90.000,E1 272.808} C_DIS
LIN {X -0.236,Y -476.346,Z 1039.513,A 0.000,B 0.000,C 90.000,E1 272.350} C_DIS
LIN {X -0.112,Y -472.029,Z 1039.510,A 0.000,B 0.000,C 90.000,E1 271.835} C_DIS
LIN {X 0.001,Y -466.838,Z 1039.507,A 0.000,B 0.000,C 90.000,E1 271.318} C_DIS
LIN {X -0.127,Y -461.118,Z 1039.505,A 0.000,B 0.000,C 90.000,E1 270.859} C_DIS
LIN {X 0.106,Y -455.021,Z 1039.502,A 0.000,B 0.000,C 90.000,E1 270.401} C_DIS
LIN {X -0.178,Y -448.377,Z 1039.500,A 0.000,B 0.000,C 90.000,E1 270.057} C_DIS
LIN {X 0.012,Y -441.009,Z 1039.498,A 0.000,B 0.000,C 90.000,E1 269.714} C_DIS
LIN {X -0.056,Y -437.298,Z 1039.498,A 0.000,B 0.000,C 90.000,E1 269.599} C_DIS
LIN {X 0.118,Y -428.939,Z 1039.497,A 0.000,B 0.000,C 90.000,E1 269.370} C_DIS
LIN {X -0.070,Y -420.409,Z 1039.496,A 0.000,B 0.000,C 90.000,E1 269.255} C_DIS
LIN {X 0.016,Y -411.605,Z 1039.495,A 0.000,B 0.000,C 90.000,E1 269.141} C_DIS
LIN {X -0.127,Y -397.510,Z 1039.495,A 0.000,B 0.000,C 90.000,E1 269.083} C_DIS
LIN {X -0.083,Y -181.332,Z 1039.495,A 0.000,B 0.000,C 90.000,E1 269.083} C_DIS
LIN {X -0.077,Y -180.905,Z 1039.474,A 0.000,B 0.000,C 90.000,E1 265.355} C_DIS
LIN {X -0.003,Y -180.669,Z 1039.469,A 0.000,B 0.000,C 90.000,E1 264.489} C_DIS
LIN {X 0.071,Y -178.750,Z 1039.441,A 0.000,B 0.000,C 90.000,E1 259.398} C_DIS
LIN {X -0.031,Y -175.798,Z 1039.413,A 0.000,B 0.000,C 90.000,E1 254.338} C_DIS
LIN {X -0.037,Y -171.983,Z 1039.384,A 0.000,B 0.000,C 90.000,E1 249.209} C_DIS
LIN {X 0.002,Y -171.389,Z 1039.380,A 0.000,B 0.000,C 90.000,E1 248.337} C_DIS
LIN {X -0.013,Y -167.632,Z 1039.356,A 0.000,B 0.000,C 90.000,E1 244.024} C_DIS
LIN {X 0.002,Y -166.289,Z 1039.346,A 0.000,B 0.000,C 90.000,E1 242.281} C_DIS
LIN {X -0.004,Y -163.037,Z 1039.327,A 0.000,B 0.000,C 90.000,E1 238.791} C_DIS
LIN {X -0.042,Y -160.967,Z 1039.312,A 0.000,B 0.000,C 90.000,E1 236.167} C_DIS
LIN {X -0.064,Y -157.719,Z 1039.292,A 0.000,B 0.000,C 90.000,E1 232.637} C_DIS
LIN {X 0.094,Y -155.758,Z 1039.277,A 0.000,B 0.000,C 90.000,E1 229.908} C_DIS
LIN {X -0.069,Y -152.015,Z 1039.253,A 0.000,B 0.000,C 90.000,E1 225.486} C_DIS
LIN {X -0.051,Y -150.262,Z 1039.238,A 0.000,B 0.000,C 90.000,E1 222.771} C_DIS
LIN {X -0.032,Y -147.016,Z 1039.212,A 0.000,B 0.000,C 90.000,E1 218.222} C_DIS
LIN {X -0.012,Y -145.599,Z 1039.197,A 0.000,B 0.000,C 90.000,E1 215.471} C_DIS
LIN {X -0.007,Y -142.985,Z 1039.172,A 0.000,B 0.000,C 90.000,E1 210.875} C_DIS
LIN {X -0.007,Y -141.612,Z 1039.151,A 0.000,B 0.000,C 90.000,E1 207.180} C_DIS
LIN {X 0.034,Y -139.427,Z 1039.115,A 0.000,B 0.000,C 90.000,E1 200.663} C_DIS
LIN {X 0.085,Y -139.157,Z 1039.104,A 0.000,B 0.000,C 90.000,E1 198.779} C_DIS
LIN {X -0.029,Y -138.342,Z 1039.058,A 0.000,B 0.000,C 90.000,E1 190.423} C_DIS
LIN {X -0.047,Y -139.481,Z 1039.006,A 0.000,B 0.000,C 90.000,E1 181.088} C_DIS
LIN {X 0.033,Y -141.073,Z 1038.975,A 0.000,B 0.000,C 90.000,E1 175.469} C_DIS
LIN {X -0.013,Y -142.449,Z 1038.959,A 0.000,B 0.000,C 90.000,E1 172.704} C_DIS
LIN {X 0.077,Y -144.690,Z 1038.934,A 0.000,B 0.000,C 90.000,E1 168.049} C_DIS
LIN {X 0.030,Y -147.282,Z 1038.913,A 0.000,B 0.000,C 90.000,E1 164.393} C_DIS
LIN {X 0.046,Y -150.601,Z 1038.888,A 0.000,B 0.000,C 90.000,E1 159.826} C_DIS
LIN {X -0.017,Y -154.074,Z 1038.868,A 0.000,B 0.000,C 90.000,E1 156.230} C_DIS
LIN {X 0.049,Y -157.494,Z 1038.848,A 0.000,B 0.000,C 90.000,E1 152.615} C_DIS
LIN {X -0.006,Y -161.721,Z 1038.828,A 0.000,B 0.000,C 90.000,E1 149.076} C_DIS
LIN {X 0.007,Y -165.915,Z 1038.809,A 0.000,B 0.000,C 90.000,E1 145.548} C_DIS
LIN {X -0.006,Y -170.902,Z 1038.789,A 0.000,B 0.000,C 90.000,E1 142.065} C_DIS
LIN {X 0.021,Y -175.770,Z 1038.770,A 0.000,B 0.000,C 90.000,E1 138.609} C_DIS
LIN {X 0.022,Y -181.380,Z 1038.751,A 0.000,B 0.000,C 90.000,E1 135.202} C_DIS
LIN {X 0.026,Y -186.874,Z 1038.732,A 0.000,B 0.000,C 90.000,E1 131.838} C_DIS
LIN {X -0.021,Y -191.459,Z 1038.719,A 0.000,B 0.000,C 90.000,E1 129.358} C_DIS
LIN {X -0.042,Y -197.599,Z 1038.700,A 0.000,B 0.000,C 90.000,E1 125.931} C_DIS
LIN {X -0.099,Y -303.506,Z 1038.699,A 0.000,B 0.000,C 90.000,E1 125.931} C_DIS
LIN {X -0.090,Y -305.636,Z 1038.699,A 0.000,B 0.000,C 90.000,E1 125.884} C_DIS
LIN {X -0.032,Y -310.988,Z 1038.698,A 0.000,B 0.000,C 90.000,E1 125.564} C_DIS
LIN {X 0.100,Y -313.906,Z 1038.696,A 0.000,B 0.000,C 90.000,E1 125.231} C_DIS
LIN {X 0.063,Y -315.930,Z 1038.694,A 0.000,B 0.000,C 90.000,E1 124.945} C_DIS
LIN {X 0.024,Y -317.515,Z 1038.693,A 0.000,B 0.000,C 90.000,E1 124.659} C_DIS
LIN {X 0.090,Y -318.896,Z 1038.691,A 0.000,B 0.000,C 90.000,E1 124.326} C_DIS
LIN {X -0.008,Y -331.262,Z 1038.671,A 0.000,B 0.000,C 90.000,E1 120.846} C_DIS
LIN {X 0.095,Y -342.801,Z 1038.656,A 0.000,B 0.000,C 90.000,E1 118.025} C_DIS
LIN {X 0.057,Y -355.777,Z 1038.641,A 0.000,B 0.000,C 90.000,E1 115.283} C_DIS
LIN {X 0.017,Y -368.605,Z 1038.627,A 0.000,B 0.000,C 90.000,E1 112.898} C_DIS
LIN {X 0.013,Y -382.746,Z 1038.614,A 0.000,B 0.000,C 90.000,E1 110.556} C_DIS
LIN {X 0.229,Y -398.300,Z 1038.601,A 0.000,B 0.000,C 90.000,E1 108.236} C_DIS
LIN {X 0.077,Y -415.379,Z 1038.589,A 0.000,B 0.000,C 90.000,E1 106.024} C_DIS
LIN {X -0.185,Y -434.103,Z 1038.577,A 0.000,B 0.000,C 90.000,E1 103.883} C_DIS
LIN {X 0.201,Y -454.069,Z 1038.566,A 0.000,B 0.000,C 90.000,E1 101.771} C_DIS
LIN {X -0.058,Y -466.822,Z 1038.559,A 0.000,B 0.000,C 90.000,E1 100.602} C_DIS
LIN {X -0.044,Y -469.015,Z 1038.558,A 0.000,B 0.000,C 90.000,E1 100.366} C_DIS
LIN {X 0.183,Y -470.794,Z 1038.556,A 0.000,B 0.000,C 90.000,E1 100.084} C_DIS
LIN {X 0.030,Y -472.131,Z 1038.555,A 0.000,B 0.000,C 90.000,E1 99.849} C_DIS
LIN {X 0.211,Y -473.803,Z 1038.552,A 0.000,B 0.000,C 90.000,E1 99.321} C_DIS
LIN {X -0.147,Y -474.408,Z 1038.549,A 0.000,B 0.000,C 90.000,E1 98.859} C_DIS
LIN {X -0.024,Y -474.050,Z 1038.546,A 0.000,B 0.000,C 90.000,E1 98.341} C_DIS
LIN {X 0.169,Y -472.676,Z 1038.544,A 0.000,B 0.000,C 90.000,E1 97.814} C_DIS
LIN {X -0.034,Y -471.540,Z 1038.542,A 0.000,B 0.000,C 90.000,E1 97.587} C_DIS
LIN {X -0.174,Y -470.025,Z 1038.541,A 0.000,B 0.000,C 90.000,E1 97.352} C_DIS
LIN {X 0.145,Y -455.862,Z 1038.529,A 0.000,B 0.000,C 90.000,E1 95.277} C_DIS
LIN {X -0.001,Y -438.212,Z 1038.515,A 0.000,B 0.000,C 90.000,E1 92.694} C_DIS
LIN {X 0.010,Y -419.159,Z 1038.497,A 0.000,B 0.000,C 90.000,E1 89.484} C_DIS
LIN {X -0.061,Y -407.518,Z 1038.485,A 0.000,B 0.000,C 90.000,E1 87.306} C_DIS
LIN {X -0.027,Y -397.116,Z 1038.474,A 0.000,B 0.000,C 90.000,E1 85.355} C_DIS
LIN {X -0.181,Y -387.942,Z 1038.465,A 0.000,B 0.000,C 90.000,E1 83.685} C_DIS
LIN {X -0.067,Y -378.594,Z 1038.455,A 0.000,B 0.000,C 90.000,E1 81.951} C_DIS
LIN {X -0.061,Y -370.529,Z 1038.447,A 0.000,B 0.000,C 90.000,E1 80.500} C_DIS
LIN {X 0.114,Y -358.939,Z 1038.436,A 0.000,B 0.000,C 90.000,E1 78.409} C_DIS
LIN {X -0.162,Y -347.347,Z 1038.424,A 0.000,B 0.000,C 90.000,E1 76.353} C_DIS
LIN {X 0.047,Y -334.284,Z 1038.410,A 0.000,B 0.000,C 90.000,E1 73.866} C_DIS
LIN {X -0.192,Y -321.720,Z 1038.396,A 0.000,B 0.000,C 90.000,E1 71.402} C_DIS
LIN {X 0.011,Y -306.595,Z 1038.379,A 0.000,B 0.000,C 90.000,E1 68.156} C_DIS
LIN {X -0.047,Y -296.345,Z 1038.366,A 0.000,B 0.000,C 90.000,E1 65.869} C_DIS
LIN {X 0.013,Y -284.904,Z 1038.351,A 0.000,B 0.000,C 90.000,E1 63.179} C_DIS
LIN {X -0.018,Y -275.097,Z 1038.338,A 0.000,B 0.000,C 90.000,E1 60.795} C_DIS
LIN {X 0.048,Y -264.096,Z 1038.322,A 0.000,B 0.000,C 90.000,E1 57.995} C_DIS
LIN {X -0.096,Y -253.373,Z 1038.306,A 0.000,B 0.000,C 90.000,E1 55.182} C_DIS
LIN {X -0.072,Y -241.795,Z 1038.288,A 0.000,B 0.000,C 90.000,E1 51.904} C_DIS
LIN {X 0.045,Y -231.015,Z 1038.270,A 0.000,B 0.000,C 90.000,E1 48.528} C_DIS
LIN {X 0.060,Y -222.042,Z 1038.253,A 0.000,B 0.000,C 90.000,E1 45.486} C_DIS
LIN {X 0.035,Y -213.560,Z 1038.236,A 0.000,B 0.000,C 90.000,E1 42.405} C_DIS
LIN {X -0.022,Y -205.596,Z 1038.218,A 0.000,B 0.000,C 90.000,E1 39.277} C_DIS
LIN {X -0.058,Y -198.135,Z 1038.200,A 0.000,B 0.000,C 90.000,E1 36.091} C_DIS
LIN {X -0.025,Y -191.267,Z 1038.182,A 0.000,B 0.000,C 90.000,E1 32.832} C_DIS
LIN {X -0.045,Y -185.131,Z 1038.164,A 0.000,B 0.000,C 90.000,E1 29.539} C_DIS
LIN {X -0.001,Y -179.747,Z 1038.145,A 0.000,B 0.000,C 90.000,E1 26.181} C_DIS
LIN {X 0.077,Y -175.181,Z 1038.127,A 0.000,B 0.000,C 90.000,E1 22.770} C_DIS
LIN {X -0.064,Y -171.318,Z 1038.108,A 0.000,B 0.000,C 90.000,E1 19.396} C_DIS
LIN {X 0.073,Y -168.209,Z 1038.089,A 0.000,B 0.000,C 90.000,E1 15.898} C_DIS
LIN {X -0.045,Y -165.287,Z 1038.064,A 0.000,B 0.000,C 90.000,E1 11.591} C_DIS
LIN {X -0.031,Y -162.916,Z 1038.030,A 0.000,B 0.000,C 90.000,E1 5.454} C_DIS
LIN {X -0.057,Y -163.898,Z 1037.963,A 0.000,B 0.000,C 90.000,E1 353.394} C_DIS
LIN {X 0.002,Y -166.607,Z 1037.934,A 0.000,B 0.000,C 90.000,E1 348.117} C_DIS
LIN {X 0.079,Y -170.039,Z 1037.910,A 0.000,B 0.000,C 90.000,E1 343.740} C_DIS
LIN {X -0.011,Y -173.498,Z 1037.891,A 0.000,B 0.000,C 90.000,E1 340.315} C_DIS
LIN {X 0.050,Y -177.664,Z 1037.872,A 0.000,B 0.000,C 90.000,E1 336.869} C_DIS
LIN {X -0.060,Y -182.666,Z 1037.853,A 0.000,B 0.000,C 90.000,E1 333.512} C_DIS
LIN {X 0.043,Y -188.528,Z 1037.834,A 0.000,B 0.000,C 90.000,E1 330.127} C_DIS
LIN {X -0.006,Y -195.198,Z 1037.816,A 0.000,B 0.000,C 90.000,E1 326.834} C_DIS
LIN {X -0.007,Y -202.572,Z 1037.798,A 0.000,B 0.000,C 90.000,E1 323.577} C_DIS
LIN {X 0.057,Y -210.442,Z 1037.780,A 0.000,B 0.000,C 90.000,E1 320.356} C_DIS
LIN {X 0.061,Y -220.082,Z 1037.760,A 0.000,B 0.000,C 90.000,E1 316.824} C_DIS
LIN {X -0.092,Y -229.483,Z 1037.743,A 0.000,B 0.000,C 90.000,E1 313.785} C_DIS
LIN {X -0.127,Y -238.616,Z 1037.728,A 0.000,B 0.000,C 90.000,E1 311.148} C_DIS
LIN {X -0.080,Y -247.625,Z 1037.716,A 0.000,B 0.000,C 90.000,E1 308.910} C_DIS
LIN {X -0.035,Y -256.131,Z 1037.706,A 0.000,B 0.000,C 90.000,E1 307.076} C_DIS
LIN {X 0.046,Y -265.574,Z 1037.696,A 0.000,B 0.000,C 90.000,E1 305.264} C_DIS
LIN {X -0.014,Y -283.963,Z 1037.678,A 0.000,B 0.000,C 90.000,E1 302.133} C_DIS
LIN {X 0.087,Y -303.872,Z 1037.662,A 0.000,B 0.000,C 90.000,E1 299.077} C_DIS
LIN {X -0.010,Y -323.062,Z 1037.647,A 0.000,B 0.000,C 90.000,E1 296.488} C_DIS
LIN {X 0.055,Y -338.677,Z 1037.637,A 0.000,B 0.000,C 90.000,E1 294.643} C_DIS
LIN {X -0.003,Y -357.725,Z 1037.626,A 0.000,B 0.000,C 90.000,E1 292.695} C_DIS
LIN {X -0.150,Y -382.661,Z 1037.613,A 0.000,B 0.000,C 90.000,E1 290.429} C_DIS
LIN {X -0.066,Y -399.181,Z 1037.605,A 0.000,B 0.000,C 90.000,E1 288.960} C_DIS
LIN {X -0.113,Y -412.605,Z 1037.599,A 0.000,B 0.000,C 90.000,E1 287.764} C_DIS
LIN {X -0.203,Y -420.425,Z 1037.594,A 0.000,B 0.000,C 90.000,E1 287.040} C_DIS
LIN {X -0.083,Y -427.939,Z 1037.590,A 0.000,B 0.000,C 90.000,E1 286.260} C_DIS
LIN {X 0.056,Y -437.757,Z 1037.584,A 0.000,B 0.000,C 90.000,E1 285.190} C_DIS
LIN {X 0.137,Y -447.009,Z 1037.578,A 0.000,B 0.000,C 90.000,E1 284.120} C_DIS
LIN {X -0.035,Y -453.411,Z 1037.574,A 0.000,B 0.000,C 90.000,E1 283.355} C_DIS
LIN {X 0.125,Y -461.117,Z 1037.568,A 0.000,B 0.000,C 90.000,E1 282.299} C_DIS
LIN {X 0.082,Y -466.274,Z 1037.564,A 0.000,B 0.000,C 90.000,E1 281.535} C_DIS
LIN {X -0.012,Y -470.848,Z 1037.560,A 0.000,B 0.000,C 90.000,E1 280.782} C_DIS
LIN {X 0.025,Y -474.742,Z 1037.556,A 0.000,B 0.000,C 90.000,E1 280.018} C_DIS
LIN {X 0.008,Y -478.161,Z 1037.552,A 0.000,B 0.000,C 90.000,E1 279.265} C_DIS
LIN {X 0.150,Y -480.134,Z 1037.549,A 0.000,B 0.000,C 90.000,E1 278.746} C_DIS
LIN {X -0.105,Y -481.807,Z 1037.546,A 0.000,B 0.000,C 90.000,E1 278.276} C_DIS
LIN {X 0.055,Y -483.269,Z 1037.543,A 0.000,B 0.000,C 90.000,E1 277.757} C_DIS
LIN {X 0.229,Y -484.499,Z 1037.540,A 0.000,B 0.000,C 90.000,E1 277.239} C_DIS
LIN {X -0.070,Y -485.524,Z 1037.538,A 0.000,B 0.000,C 90.000,E1 276.777} C_DIS
LIN {X 0.120,Y -486.294,Z 1037.535,A 0.000,B 0.000,C 90.000,E1 276.258} C_DIS
LIN {X -0.167,Y -486.810,Z 1037.532,A 0.000,B 0.000,C 90.000,E1 275.796} C_DIS
LIN {X 0.032,Y -486.929,Z 1037.529,A 0.000,B 0.000,C 90.000,E1 275.277} C_DIS
LIN {X 0.233,Y -486.620,Z 1037.527,A 0.000,B 0.000,C 90.000,E1 274.759} C_DIS
LIN {X -0.088,Y -485.855,Z 1037.524,A 0.000,B 0.000,C 90.000,E1 274.302} C_DIS
LIN {X 0.110,Y -484.500,Z 1037.521,A 0.000,B 0.000,C 90.000,E1 273.784} C_DIS
LIN {X -0.211,Y -482.576,Z 1037.518,A 0.000,B 0.000,C 90.000,E1 273.326} C_DIS
LIN {X -0.029,Y -479.904,Z 1037.516,A 0.000,B 0.000,C 90.000,E1 272.808} C_DIS
LIN {X 0.110,Y -476.439,Z 1037.513,A 0.000,B 0.000,C 90.000,E1 272.293} C_DIS
LIN {X -0.226,Y -472.162,Z 1037.510,A 0.000,B 0.000,C 90.000,E1 271.833} C_DIS
LIN {X -0.125,Y -466.984,Z 1037.507,A 0.000,B 0.000,C 90.000,E1 271.318} C_DIS
LIN {X 0.219,Y -461.285,Z 1037.505,A 0.000,B 0.000,C 90.000,E1 270.802} C_DIS
LIN {X -0.028,Y -455.136,Z 1037.502,A 0.000,B 0.000,C 90.000,E1 270.401} C_DIS
LIN {X 0.156,Y -448.523,Z 1037.500,A 0.000,B 0.000,C 90.000,E1 270.000} C_DIS
LIN {X -0.112,Y -441.066,Z 1037.498,A 0.000,B 0.000,C 90.000,E1 269.714} C_DIS
LIN {X -0.176,Y -437.353,Z 1037.498,A 0.000,B 0.000,C 90.000,E1 269.599} C_DIS
LIN {X -0.005,Y -428.983,Z 1037.496,A 0.000,B 0.000,C 90.000,E1 269.370} C_DIS
LIN {X -0.197,Y -420.269,Z 1037.496,A 0.000,B 0.000,C 90.000,E1 269.255} C_DIS
LIN {X -0.090,Y -411.336,Z 1037.495,A 0.000,B 0.000,C 90.000,E1 269.141} C_DIS
LIN {X 0.126,Y -395.713,Z 1037.495,A 0.000,B 0.000,C 90.000,E1 269.026} C_DIS
LIN {X 0.032,Y -181.327,Z 1037.495,A 0.000,B 0.000,C 90.000,E1 269.026} C_DIS
LIN {X 0.063,Y -180.905,Z 1037.474,A 0.000,B 0.000,C 90.000,E1 265.298} C_DIS
LIN {X 0.013,Y -180.253,Z 1037.465,A 0.000,B 0.000,C 90.000,E1 263.628} C_DIS
LIN {X 0.032,Y -178.743,Z 1037.441,A 0.000,B 0.000,C 90.000,E1 259.398} C_DIS
LIN {X -0.071,Y -175.790,Z 1037.413,A 0.000,B 0.000,C 90.000,E1 254.338} C_DIS
LIN {X -0.075,Y -171.975,Z 1037.384,A 0.000,B 0.000,C 90.000,E1 249.209} C_DIS
LIN {X -0.037,Y -171.377,Z 1037.380,A 0.000,B 0.000,C 90.000,E1 248.337} C_DIS
LIN {X -0.052,Y -167.623,Z 1037.356,A 0.000,B 0.000,C 90.000,E1 244.024} C_DIS
LIN {X -0.036,Y -166.275,Z 1037.346,A 0.000,B 0.000,C 90.000,E1 242.281} C_DIS
LIN {X -0.041,Y -163.026,Z 1037.327,A 0.000,B 0.000,C 90.000,E1 238.791} C_DIS
LIN {X 0.010,Y -160.954,Z 1037.312,A 0.000,B 0.000,C 90.000,E1 236.135} C_DIS
LIN {X -0.006,Y -157.709,Z 1037.292,A 0.000,B 0.000,C 90.000,E1 232.603} C_DIS
LIN {X 0.058,Y -155.749,Z 1037.277,A 0.000,B 0.000,C 90.000,E1 229.908} C_DIS
LIN {X 0.003,Y -152.004,Z 1037.252,A 0.000,B 0.000,C 90.000,E1 225.445} C_DIS
LIN {X -0.087,Y -150.251,Z 1037.237,A 0.000,B 0.000,C 90.000,E1 222.771} C_DIS
LIN {X 0.048,Y -147.007,Z 1037.212,A 0.000,B 0.000,C 90.000,E1 218.177} C_DIS
LIN {X 0.037,Y -145.591,Z 1037.197,A 0.000,B 0.000,C 90.000,E1 215.438} C_DIS
LIN {X -0.041,Y -142.979,Z 1037.171,A 0.000,B 0.000,C 90.000,E1 210.875} C_DIS
LIN {X -0.042,Y -141.605,Z 1037.151,A 0.000,B 0.000,C 90.000,E1 207.180} C_DIS
LIN {X 0.000,Y -139.425,Z 1037.115,A 0.000,B 0.000,C 90.000,E1 200.663} C_DIS
LIN {X 0.050,Y -139.154,Z 1037.104,A 0.000,B 0.000,C 90.000,E1 198.779} C_DIS
LIN {X 0.072,Y -138.344,Z 1037.058,A 0.000,B 0.000,C 90.000,E1 190.366} C_DIS
LIN {X 0.059,Y -139.484,Z 1037.006,A 0.000,B 0.000,C 90.000,E1 181.031} C_DIS
LIN {X -0.001,Y -141.079,Z 1036.975,A 0.000,B 0.000,C 90.000,E1 175.469} C_DIS
LIN {X -0.047,Y -142.455,Z 1036.959,A 0.000,B 0.000,C 90.000,E1 172.704} C_DIS
LIN {X 0.042,Y -144.698,Z 1036.934,A 0.000,B 0.000,C 90.000,E1 168.049} C_DIS
LIN {X -0.005,Y -147.293,Z 1036.913,A 0.000,B 0.000,C 90.000,E1 164.393} C_DIS
LIN {X 0.011,Y -150.612,Z 1036.888,A 0.000,B 0.000,C 90.000,E1 159.826} C_DIS
LIN {X -0.054,Y -154.087,Z 1036.868,A 0.000,B 0.000,C 90.000,E1 156.230} C_DIS
LIN {X 0.012,Y -157.508,Z 1036.848,A 0.000,B 0.000,C 90.000,E1 152.615} C_DIS
LIN {X -0.043,Y -161.739,Z 1036.828,A 0.000,B 0.000,C 90.000,E1 149.076} C_DIS
END
